// TwinCAT 3 PLC project TF3820StandalonePLC
// ProgramVersion: 3.1.4026.20
// libraries:
//   Tc2_Standard, * (Beckhoff Automation GmbH)
//   Tc2_System, * (Beckhoff Automation GmbH)
//   Tc3_MlServer, * (Beckhoff Automation GmbH)
// project tree:
//   DUTs/ E_TF3820StandaloneModelId.TcDUT, ST_FeedforwardInput.TcDUT, ST_FeedforwardOutput.TcDUT, ST_GruSequenceInput.TcDUT, ST_GruSequenceOutput.TcDUT, ST_HarmonicRegressionInput.TcDUT, ST_HarmonicRegressionOutput.TcDUT, ST_LstmSequenceInput.TcDUT, ST_LstmSequenceOutput.TcDUT, ST_PeriodicGruSequenceInput.TcDUT, ST_PeriodicGruSequenceOutput.TcDUT, ST_PeriodicLstmSequenceInput.TcDUT, ST_PeriodicLstmSequenceOutput.TcDUT, ST_PeriodicMlpInput.TcDUT, ST_PeriodicMlpOutput.TcDUT, ST_PeriodicMlpHarmonicInput.TcDUT, ST_PeriodicMlpHarmonicOutput.TcDUT, ST_PeriodicTemporalConvolutionInput.TcDUT, ST_PeriodicTemporalConvolutionOutput.TcDUT, ST_RcimTrack1Input.TcDUT, ST_RcimTrack1Output.TcDUT, ST_ResidualHarmonicGruSequenceDense240Input.TcDUT, ST_ResidualHarmonicGruSequenceDense240Output.TcDUT, ST_ResidualHarmonicGruSequenceDense360Input.TcDUT, ST_ResidualHarmonicGruSequenceDense360Output.TcDUT, ST_ResidualHarmonicGruSequenceSparseRcimInput.TcDUT, ST_ResidualHarmonicGruSequenceSparseRcimOutput.TcDUT, ST_ResidualHarmonicLstmSequenceDense240Input.TcDUT, ST_ResidualHarmonicLstmSequenceDense240Output.TcDUT, ST_ResidualHarmonicLstmSequenceDense360Input.TcDUT, ST_ResidualHarmonicLstmSequenceDense360Output.TcDUT, ST_ResidualHarmonicLstmSequenceSparseRcimInput.TcDUT, ST_ResidualHarmonicLstmSequenceSparseRcimOutput.TcDUT, ST_ResidualHarmonicMlpInput.TcDUT, ST_ResidualHarmonicMlpOutput.TcDUT, ST_TemporalConvolutionInput.TcDUT, ST_TemporalConvolutionOutput.TcDUT, ST_TreeInput.TcDUT, ST_TreeOutput.TcDUT, ST_Wave31SequentialResidualOffsetProbeInput.TcDUT, ST_Wave31SequentialResidualOffsetProbeOutput.TcDUT, ST_Wave32CleanSequentialResidualOffsetInput.TcDUT, ST_Wave32CleanSequentialResidualOffsetOutput.TcDUT, ST_Wave32HarmonicResidualOffsetInput.TcDUT, ST_Wave32HarmonicResidualOffsetOutput.TcDUT, ST_Wave33CurveAwarePointwiseControlInput.TcDUT, ST_Wave33CurveAwarePointwiseControlOutput.TcDUT, ST_Wave33FullCurveCompositeInput.TcDUT, ST_Wave33FullCurveCompositeOutput.TcDUT, ST_Wave33RawCenteredShapeCurveAwareInput.TcDUT, ST_Wave33RawCenteredShapeCurveAwareOutput.TcDUT, ST_Wave33RawOffsetCurveAwareInput.TcDUT, ST_Wave33RawOffsetCurveAwareOutput.TcDUT, ST_Wave41LogCoshRobustLossInput.TcDUT, ST_Wave41LogCoshRobustLossOutput.TcDUT, ST_Wave41MaeRobustLossInput.TcDUT, ST_Wave41MaeRobustLossOutput.TcDUT, ST_Wave41SmoothL1RobustLossInput.TcDUT, ST_Wave41SmoothL1RobustLossOutput.TcDUT, ST_Wave42GaussianNllInput.TcDUT, ST_Wave42GaussianNllOutput.TcDUT, ST_Wave42QuantileP10P50P90Input.TcDUT, ST_Wave42QuantileP10P50P90Output.TcDUT, ST_Wave43MixtureDensityK2Input.TcDUT, ST_Wave43MixtureDensityK2Output.TcDUT, ST_Wave43MixtureDensityK3Input.TcDUT, ST_Wave43MixtureDensityK3Output.TcDUT, ST_Wave44CausalTcnLatentOffsetResidualInput.TcDUT, ST_Wave44CausalTcnLatentOffsetResidualOutput.TcDUT, ST_Wave44GruLatentOffsetResidualInput.TcDUT, ST_Wave44GruLatentOffsetResidualOutput.TcDUT, ST_Wave51HarmonicPriorPointwiseControlInput.TcDUT, ST_Wave51HarmonicPriorPointwiseControlOutput.TcDUT, ST_Wave51HarmonicPriorSmoothL1StructuredInput.TcDUT, ST_Wave51HarmonicPriorSmoothL1StructuredOutput.TcDUT
//   / PlcTask_TF3820Standalone.TcTTO
//   POUs/ FB_FeedforwardTf3820Runner.TcPOU, FB_GruSequenceTf3820Runner.TcPOU, FB_HarmonicRegressionTf3820Runner.TcPOU, FB_LstmSequenceTf3820Runner.TcPOU, FB_PeriodicGruSequenceTf3820Runner.TcPOU, FB_PeriodicLstmSequenceTf3820Runner.TcPOU, FB_PeriodicMlpTf3820Runner.TcPOU, FB_PeriodicMlpHarmonicTf3820Runner.TcPOU, FB_PeriodicTemporalConvolutionTf3820Runner.TcPOU, FB_RcimTrack1Tf3820Runner.TcPOU, FB_ResidualHarmonicGruSequenceDense240Tf3820Runner.TcPOU, FB_ResidualHarmonicGruSequenceDense360Tf3820Runner.TcPOU, FB_ResidualHarmonicGruSequenceSparseRcimTf3820Runner.TcPOU, FB_ResidualHarmonicLstmSequenceDense240Tf3820Runner.TcPOU, FB_ResidualHarmonicLstmSequenceDense360Tf3820Runner.TcPOU, FB_ResidualHarmonicLstmSequenceSparseRcimTf3820Runner.TcPOU, FB_ResidualHarmonicMlpTf3820Runner.TcPOU, FB_TemporalConvolutionTf3820Runner.TcPOU, FB_TreeTf3820Runner.TcPOU, FB_Wave31SequentialResidualOffsetProbeTf3820Runner.TcPOU, FB_Wave32CleanSequentialResidualOffsetTf3820Runner.TcPOU, FB_Wave32HarmonicResidualOffsetTf3820Runner.TcPOU, FB_Wave33CurveAwarePointwiseControlTf3820Runner.TcPOU, FB_Wave33FullCurveCompositeTf3820Runner.TcPOU, FB_Wave33RawCenteredShapeCurveAwareTf3820Runner.TcPOU, FB_Wave33RawOffsetCurveAwareTf3820Runner.TcPOU, FB_Wave41LogCoshRobustLossTf3820Runner.TcPOU, FB_Wave41MaeRobustLossTf3820Runner.TcPOU, FB_Wave41SmoothL1RobustLossTf3820Runner.TcPOU, FB_Wave42GaussianNllTf3820Runner.TcPOU, FB_Wave42QuantileP10P50P90Tf3820Runner.TcPOU, FB_Wave43MixtureDensityK2Tf3820Runner.TcPOU, FB_Wave43MixtureDensityK3Tf3820Runner.TcPOU, FB_Wave44CausalTcnLatentOffsetResidualTf3820Runner.TcPOU, FB_Wave44GruLatentOffsetResidualTf3820Runner.TcPOU, FB_Wave51HarmonicPriorPointwiseControlTf3820Runner.TcPOU, FB_Wave51HarmonicPriorSmoothL1StructuredTf3820Runner.TcPOU, P_TF3820StandaloneModelTest.TcPOU
// real-time tasks:
//   TASK PlcTask_TF3820Standalone: cycle T#1ms, priority 10, ADS port 350

CONFIGURATION TF3820StandalonePLC
    RESOURCE PLC ON TwinCAT3
        TASK PlcTask_TF3820Standalone(INTERVAL := T#1ms, PRIORITY := 10);
        PROGRAM P_TF3820StandaloneModelTest WITH PlcTask_TF3820Standalone : P_TF3820StandaloneModelTest;
    END_RESOURCE
END_CONFIGURATION

// ---- DUTs/E_TF3820StandaloneModelId.TcDUT
{attribute 'qualified_only'}
{attribute 'strict'}
TYPE E_TF3820StandaloneModelId :
(
	Model_Feedforward := 0,
	Model_Gru_Sequence := 1,
	Model_Harmonic_Regression := 2,
	Model_Lstm_Sequence := 3,
	Model_Periodic_Gru_Sequence := 4,
	Model_Periodic_Lstm_Sequence := 5,
	Model_Periodic_Mlp := 6,
	Model_Periodic_Mlp_Harmonic := 7,
	Model_Periodic_Temporal_Convolution := 8,
	Model_Rcim_Track1 := 9,
	Model_Residual_Harmonic_Gru_Sequence_Dense240 := 10,
	Model_Residual_Harmonic_Gru_Sequence_Dense360 := 11,
	Model_Residual_Harmonic_Gru_Sequence_Sparse_Rcim := 12,
	Model_Residual_Harmonic_Lstm_Sequence_Dense240 := 13,
	Model_Residual_Harmonic_Lstm_Sequence_Dense360 := 14,
	Model_Residual_Harmonic_Lstm_Sequence_Sparse_Rcim := 15,
	Model_Residual_Harmonic_Mlp := 16,
	Model_Temporal_Convolution := 17,
	Model_Tree := 18,
	Model_Wave3_1_Sequential_Residual_Offset_Probe := 19,
	Model_Wave3_2_Clean_Sequential_Residual_Offset := 20,
	Model_Wave3_2_Harmonic_Residual_Offset := 21,
	Model_Wave3_3_Curve_Aware_Pointwise_Control := 22,
	Model_Wave3_3_Full_Curve_Composite := 23,
	Model_Wave3_3_Raw_Centered_Shape_Curve_Aware := 24,
	Model_Wave3_3_Raw_Offset_Curve_Aware := 25,
	Model_Wave4_1_Log_Cosh_Robust_Loss := 26,
	Model_Wave4_1_Mae_Robust_Loss := 27,
	Model_Wave4_1_Smooth_L1_Robust_Loss := 28,
	Model_Wave4_2_Gaussian_Nll := 29,
	Model_Wave4_2_Quantile_P10_P50_P90 := 30,
	Model_Wave4_3_Mixture_Density_K2 := 31,
	Model_Wave4_3_Mixture_Density_K3 := 32,
	Model_Wave4_4_Causal_Tcn_Latent_Offset_Residual := 33,
	Model_Wave4_4_Gru_Latent_Offset_Residual := 34,
	Model_Wave5_1_Harmonic_Prior_Pointwise_Control := 35,
	Model_Wave5_1_Harmonic_Prior_Smooth_L1_Structured := 36
);
END_TYPE

// ---- DUTs/ST_FeedforwardInput.TcDUT
TYPE ST_FeedforwardInput :
STRUCT

	{attribute 'hide'} _header_DO_NOT_CHANGE : ARRAY[0..63] OF SINT := [-1,-112,120,86,52,18,-1,-1,1,-1,0,0,-1,-1,-112,-112,61,-49,110,-13,101,63,-28,35,-75,-48,62,84,75,113,93,86,13,-100,61,-11,-76,-124,91,74,-32,110,127,-106,67,10,-85,-84,84,0,0,0,0,0,0,0,0,0,0,0,0,0,0,0];
	in_input_tensor : ARRAY[0..0,0..4] OF REAL;

END_STRUCT
END_TYPE

// ---- DUTs/ST_FeedforwardOutput.TcDUT
TYPE ST_FeedforwardOutput :
STRUCT

	{attribute 'hide'} _header_DO_NOT_CHANGE : ARRAY[0..63] OF SINT := [-1,-112,120,86,52,18,-1,-1,1,-1,0,0,-1,-1,-112,-112,-35,24,-50,75,-65,96,-121,123,127,87,61,127,-39,-108,16,-70,120,-89,-28,78,-43,26,-32,-7,81,19,29,-89,-55,3,43,2,68,0,0,0,0,0,0,0,0,0,0,0,0,0,0,0];
	out_prediction_tensor : ARRAY[0..0,0..0] OF REAL;

END_STRUCT
END_TYPE

// ---- DUTs/ST_GruSequenceInput.TcDUT
TYPE ST_GruSequenceInput :
STRUCT

	{attribute 'hide'} _header_DO_NOT_CHANGE : ARRAY[0..63] OF SINT := [-1,-112,120,86,52,18,-1,-1,1,-1,0,0,-1,-1,-112,-112,76,-37,-101,-100,-56,125,72,-20,-8,-106,39,-43,33,76,57,117,-100,-22,-66,-55,64,-24,-107,-56,26,-38,-68,-13,105,114,16,-98,-44,2,0,0,0,0,0,0,0,0,0,0,0,0,0,0];
	in_input_tensor : ARRAY[0..0,0..32,0..4] OF REAL;

END_STRUCT
END_TYPE

// ---- DUTs/ST_GruSequenceOutput.TcDUT
TYPE ST_GruSequenceOutput :
STRUCT

	{attribute 'hide'} _header_DO_NOT_CHANGE : ARRAY[0..63] OF SINT := [-1,-112,120,86,52,18,-1,-1,1,-1,0,0,-1,-1,-112,-112,-35,24,-50,75,-65,96,-121,123,127,87,61,127,-39,-108,16,-70,120,-89,-28,78,-43,26,-32,-7,81,19,29,-89,-55,3,43,2,68,0,0,0,0,0,0,0,0,0,0,0,0,0,0,0];
	out_prediction_tensor : ARRAY[0..0,0..0] OF REAL;

END_STRUCT
END_TYPE

// ---- DUTs/ST_HarmonicRegressionInput.TcDUT
TYPE ST_HarmonicRegressionInput :
STRUCT

	{attribute 'hide'} _header_DO_NOT_CHANGE : ARRAY[0..63] OF SINT := [-1,-112,120,86,52,18,-1,-1,1,-1,0,0,-1,-1,-112,-112,61,-49,110,-13,101,63,-28,35,-75,-48,62,84,75,113,93,86,13,-100,61,-11,-76,-124,91,74,-32,110,127,-106,67,10,-85,-84,84,0,0,0,0,0,0,0,0,0,0,0,0,0,0,0];
	in_input_tensor : ARRAY[0..0,0..4] OF REAL;

END_STRUCT
END_TYPE

// ---- DUTs/ST_HarmonicRegressionOutput.TcDUT
TYPE ST_HarmonicRegressionOutput :
STRUCT

	{attribute 'hide'} _header_DO_NOT_CHANGE : ARRAY[0..63] OF SINT := [-1,-112,120,86,52,18,-1,-1,1,-1,0,0,-1,-1,-112,-112,-35,24,-50,75,-65,96,-121,123,127,87,61,127,-39,-108,16,-70,120,-89,-28,78,-43,26,-32,-7,81,19,29,-89,-55,3,43,2,68,0,0,0,0,0,0,0,0,0,0,0,0,0,0,0];
	out_prediction_tensor : ARRAY[0..0,0..0] OF REAL;

END_STRUCT
END_TYPE

// ---- DUTs/ST_LstmSequenceInput.TcDUT
TYPE ST_LstmSequenceInput :
STRUCT

	{attribute 'hide'} _header_DO_NOT_CHANGE : ARRAY[0..63] OF SINT := [-1,-112,120,86,52,18,-1,-1,1,-1,0,0,-1,-1,-112,-112,76,-37,-101,-100,-56,125,72,-20,-8,-106,39,-43,33,76,57,117,-100,-22,-66,-55,64,-24,-107,-56,26,-38,-68,-13,105,114,16,-98,-44,2,0,0,0,0,0,0,0,0,0,0,0,0,0,0];
	in_input_tensor : ARRAY[0..0,0..32,0..4] OF REAL;

END_STRUCT
END_TYPE

// ---- DUTs/ST_LstmSequenceOutput.TcDUT
TYPE ST_LstmSequenceOutput :
STRUCT

	{attribute 'hide'} _header_DO_NOT_CHANGE : ARRAY[0..63] OF SINT := [-1,-112,120,86,52,18,-1,-1,1,-1,0,0,-1,-1,-112,-112,-35,24,-50,75,-65,96,-121,123,127,87,61,127,-39,-108,16,-70,120,-89,-28,78,-43,26,-32,-7,81,19,29,-89,-55,3,43,2,68,0,0,0,0,0,0,0,0,0,0,0,0,0,0,0];
	out_prediction_tensor : ARRAY[0..0,0..0] OF REAL;

END_STRUCT
END_TYPE

// ---- DUTs/ST_PeriodicGruSequenceInput.TcDUT
TYPE ST_PeriodicGruSequenceInput :
STRUCT

	{attribute 'hide'} _header_DO_NOT_CHANGE : ARRAY[0..63] OF SINT := [-1,-112,120,86,52,18,-1,-1,1,-1,0,0,-1,-1,-112,-112,76,-37,-101,-100,-56,125,72,-20,-8,-106,39,-43,33,76,57,117,-100,-22,-66,-55,64,-24,-107,-56,26,-38,-68,-13,105,114,16,-98,-44,2,0,0,0,0,0,0,0,0,0,0,0,0,0,0];
	in_input_tensor : ARRAY[0..0,0..32,0..4] OF REAL;

END_STRUCT
END_TYPE

// ---- DUTs/ST_PeriodicGruSequenceOutput.TcDUT
TYPE ST_PeriodicGruSequenceOutput :
STRUCT

	{attribute 'hide'} _header_DO_NOT_CHANGE : ARRAY[0..63] OF SINT := [-1,-112,120,86,52,18,-1,-1,1,-1,0,0,-1,-1,-112,-112,-35,24,-50,75,-65,96,-121,123,127,87,61,127,-39,-108,16,-70,120,-89,-28,78,-43,26,-32,-7,81,19,29,-89,-55,3,43,2,68,0,0,0,0,0,0,0,0,0,0,0,0,0,0,0];
	out_prediction_tensor : ARRAY[0..0,0..0] OF REAL;

END_STRUCT
END_TYPE

// ---- DUTs/ST_PeriodicLstmSequenceInput.TcDUT
TYPE ST_PeriodicLstmSequenceInput :
STRUCT

	{attribute 'hide'} _header_DO_NOT_CHANGE : ARRAY[0..63] OF SINT := [-1,-112,120,86,52,18,-1,-1,1,-1,0,0,-1,-1,-112,-112,76,-37,-101,-100,-56,125,72,-20,-8,-106,39,-43,33,76,57,117,-100,-22,-66,-55,64,-24,-107,-56,26,-38,-68,-13,105,114,16,-98,-44,2,0,0,0,0,0,0,0,0,0,0,0,0,0,0];
	in_input_tensor : ARRAY[0..0,0..32,0..4] OF REAL;

END_STRUCT
END_TYPE

// ---- DUTs/ST_PeriodicLstmSequenceOutput.TcDUT
TYPE ST_PeriodicLstmSequenceOutput :
STRUCT

	{attribute 'hide'} _header_DO_NOT_CHANGE : ARRAY[0..63] OF SINT := [-1,-112,120,86,52,18,-1,-1,1,-1,0,0,-1,-1,-112,-112,-35,24,-50,75,-65,96,-121,123,127,87,61,127,-39,-108,16,-70,120,-89,-28,78,-43,26,-32,-7,81,19,29,-89,-55,3,43,2,68,0,0,0,0,0,0,0,0,0,0,0,0,0,0,0];
	out_prediction_tensor : ARRAY[0..0,0..0] OF REAL;

END_STRUCT
END_TYPE

// ---- DUTs/ST_PeriodicMlpInput.TcDUT
TYPE ST_PeriodicMlpInput :
STRUCT

	{attribute 'hide'} _header_DO_NOT_CHANGE : ARRAY[0..63] OF SINT := [-1,-112,120,86,52,18,-1,-1,1,-1,0,0,-1,-1,-112,-112,61,-49,110,-13,101,63,-28,35,-75,-48,62,84,75,113,93,86,13,-100,61,-11,-76,-124,91,74,-32,110,127,-106,67,10,-85,-84,84,0,0,0,0,0,0,0,0,0,0,0,0,0,0,0];
	in_input_tensor : ARRAY[0..0,0..4] OF REAL;

END_STRUCT
END_TYPE

// ---- DUTs/ST_PeriodicMlpOutput.TcDUT
TYPE ST_PeriodicMlpOutput :
STRUCT

	{attribute 'hide'} _header_DO_NOT_CHANGE : ARRAY[0..63] OF SINT := [-1,-112,120,86,52,18,-1,-1,1,-1,0,0,-1,-1,-112,-112,-35,24,-50,75,-65,96,-121,123,127,87,61,127,-39,-108,16,-70,120,-89,-28,78,-43,26,-32,-7,81,19,29,-89,-55,3,43,2,68,0,0,0,0,0,0,0,0,0,0,0,0,0,0,0];
	out_prediction_tensor : ARRAY[0..0,0..0] OF REAL;

END_STRUCT
END_TYPE

// ---- DUTs/ST_PeriodicMlpHarmonicInput.TcDUT
TYPE ST_PeriodicMlpHarmonicInput :
STRUCT

	{attribute 'hide'} _header_DO_NOT_CHANGE : ARRAY[0..63] OF SINT := [-1,-112,120,86,52,18,-1,-1,1,-1,0,0,-1,-1,-112,-112,61,-49,110,-13,101,63,-28,35,-75,-48,62,84,75,113,93,86,13,-100,61,-11,-76,-124,91,74,-32,110,127,-106,67,10,-85,-84,84,0,0,0,0,0,0,0,0,0,0,0,0,0,0,0];
	in_input_tensor : ARRAY[0..0,0..4] OF REAL;

END_STRUCT
END_TYPE

// ---- DUTs/ST_PeriodicMlpHarmonicOutput.TcDUT
TYPE ST_PeriodicMlpHarmonicOutput :
STRUCT

	{attribute 'hide'} _header_DO_NOT_CHANGE : ARRAY[0..63] OF SINT := [-1,-112,120,86,52,18,-1,-1,1,-1,0,0,-1,-1,-112,-112,-35,24,-50,75,-65,96,-121,123,127,87,61,127,-39,-108,16,-70,120,-89,-28,78,-43,26,-32,-7,81,19,29,-89,-55,3,43,2,68,0,0,0,0,0,0,0,0,0,0,0,0,0,0,0];
	out_prediction_tensor : ARRAY[0..0,0..0] OF REAL;

END_STRUCT
END_TYPE

// ---- DUTs/ST_PeriodicTemporalConvolutionInput.TcDUT
TYPE ST_PeriodicTemporalConvolutionInput :
STRUCT

	{attribute 'hide'} _header_DO_NOT_CHANGE : ARRAY[0..63] OF SINT := [-1,-112,120,86,52,18,-1,-1,1,-1,0,0,-1,-1,-112,-112,76,-37,-101,-100,-56,125,72,-20,-8,-106,39,-43,33,76,57,117,-100,-22,-66,-55,64,-24,-107,-56,26,-38,-68,-13,105,114,16,-98,-44,2,0,0,0,0,0,0,0,0,0,0,0,0,0,0];
	in_input_tensor : ARRAY[0..0,0..32,0..4] OF REAL;

END_STRUCT
END_TYPE

// ---- DUTs/ST_PeriodicTemporalConvolutionOutput.TcDUT
TYPE ST_PeriodicTemporalConvolutionOutput :
STRUCT

	{attribute 'hide'} _header_DO_NOT_CHANGE : ARRAY[0..63] OF SINT := [-1,-112,120,86,52,18,-1,-1,1,-1,0,0,-1,-1,-112,-112,-35,24,-50,75,-65,96,-121,123,127,87,61,127,-39,-108,16,-70,120,-89,-28,78,-43,26,-32,-7,81,19,29,-89,-55,3,43,2,68,0,0,0,0,0,0,0,0,0,0,0,0,0,0,0];
	out_prediction_tensor : ARRAY[0..0,0..0] OF REAL;

END_STRUCT
END_TYPE

// ---- DUTs/ST_RcimTrack1Input.TcDUT
TYPE ST_RcimTrack1Input :
STRUCT

	{attribute 'hide'} _header_DO_NOT_CHANGE : ARRAY[0..63] OF SINT := [-1,-112,120,86,52,18,-1,-1,1,-1,0,0,-1,-1,-112,-112,65,64,108,85,118,21,-37,1,110,122,-102,19,93,-117,-35,-43,3,-45,33,-52,25,-24,90,7,83,36,22,5,-43,-65,-103,-61,76,0,0,0,0,0,0,0,0,0,0,0,0,0,0,0];
	in_float_input : ARRAY[0..0,0..2] OF REAL;

END_STRUCT
END_TYPE

// ---- DUTs/ST_RcimTrack1Output.TcDUT
TYPE ST_RcimTrack1Output :
STRUCT

	{attribute 'hide'} _header_DO_NOT_CHANGE : ARRAY[0..63] OF SINT := [-1,-112,120,86,52,18,-1,-1,1,-1,0,0,-1,-1,-112,-112,-35,24,-50,75,-65,96,-121,123,127,87,61,127,-39,-108,16,-70,120,-89,-28,78,-43,26,-32,-7,81,19,29,-89,-55,3,43,2,68,0,0,0,0,0,0,0,0,0,0,0,0,0,0,0];
	out_variable : ARRAY[0..0,0..0] OF REAL;

END_STRUCT
END_TYPE

// ---- DUTs/ST_ResidualHarmonicGruSequenceDense240Input.TcDUT
TYPE ST_ResidualHarmonicGruSequenceDense240Input :
STRUCT

	{attribute 'hide'} _header_DO_NOT_CHANGE : ARRAY[0..63] OF SINT := [-1,-112,120,86,52,18,-1,-1,1,-1,0,0,-1,-1,-112,-112,76,-37,-101,-100,-56,125,72,-20,-8,-106,39,-43,33,76,57,117,-100,-22,-66,-55,64,-24,-107,-56,26,-38,-68,-13,105,114,16,-98,-44,2,0,0,0,0,0,0,0,0,0,0,0,0,0,0];
	in_input_tensor : ARRAY[0..0,0..32,0..4] OF REAL;

END_STRUCT
END_TYPE

// ---- DUTs/ST_ResidualHarmonicGruSequenceDense240Output.TcDUT
TYPE ST_ResidualHarmonicGruSequenceDense240Output :
STRUCT

	{attribute 'hide'} _header_DO_NOT_CHANGE : ARRAY[0..63] OF SINT := [-1,-112,120,86,52,18,-1,-1,1,-1,0,0,-1,-1,-112,-112,-35,24,-50,75,-65,96,-121,123,127,87,61,127,-39,-108,16,-70,120,-89,-28,78,-43,26,-32,-7,81,19,29,-89,-55,3,43,2,68,0,0,0,0,0,0,0,0,0,0,0,0,0,0,0];
	out_prediction_tensor : ARRAY[0..0,0..0] OF REAL;

END_STRUCT
END_TYPE

// ---- DUTs/ST_ResidualHarmonicGruSequenceDense360Input.TcDUT
TYPE ST_ResidualHarmonicGruSequenceDense360Input :
STRUCT

	{attribute 'hide'} _header_DO_NOT_CHANGE : ARRAY[0..63] OF SINT := [-1,-112,120,86,52,18,-1,-1,1,-1,0,0,-1,-1,-112,-112,76,-37,-101,-100,-56,125,72,-20,-8,-106,39,-43,33,76,57,117,-100,-22,-66,-55,64,-24,-107,-56,26,-38,-68,-13,105,114,16,-98,-44,2,0,0,0,0,0,0,0,0,0,0,0,0,0,0];
	in_input_tensor : ARRAY[0..0,0..32,0..4] OF REAL;

END_STRUCT
END_TYPE

// ---- DUTs/ST_ResidualHarmonicGruSequenceDense360Output.TcDUT
TYPE ST_ResidualHarmonicGruSequenceDense360Output :
STRUCT

	{attribute 'hide'} _header_DO_NOT_CHANGE : ARRAY[0..63] OF SINT := [-1,-112,120,86,52,18,-1,-1,1,-1,0,0,-1,-1,-112,-112,-35,24,-50,75,-65,96,-121,123,127,87,61,127,-39,-108,16,-70,120,-89,-28,78,-43,26,-32,-7,81,19,29,-89,-55,3,43,2,68,0,0,0,0,0,0,0,0,0,0,0,0,0,0,0];
	out_prediction_tensor : ARRAY[0..0,0..0] OF REAL;

END_STRUCT
END_TYPE

// ---- DUTs/ST_ResidualHarmonicGruSequenceSparseRcimInput.TcDUT
TYPE ST_ResidualHarmonicGruSequenceSparseRcimInput :
STRUCT

	{attribute 'hide'} _header_DO_NOT_CHANGE : ARRAY[0..63] OF SINT := [-1,-112,120,86,52,18,-1,-1,1,-1,0,0,-1,-1,-112,-112,76,-37,-101,-100,-56,125,72,-20,-8,-106,39,-43,33,76,57,117,-100,-22,-66,-55,64,-24,-107,-56,26,-38,-68,-13,105,114,16,-98,-44,2,0,0,0,0,0,0,0,0,0,0,0,0,0,0];
	in_input_tensor : ARRAY[0..0,0..32,0..4] OF REAL;

END_STRUCT
END_TYPE

// ---- DUTs/ST_ResidualHarmonicGruSequenceSparseRcimOutput.TcDUT
TYPE ST_ResidualHarmonicGruSequenceSparseRcimOutput :
STRUCT

	{attribute 'hide'} _header_DO_NOT_CHANGE : ARRAY[0..63] OF SINT := [-1,-112,120,86,52,18,-1,-1,1,-1,0,0,-1,-1,-112,-112,-35,24,-50,75,-65,96,-121,123,127,87,61,127,-39,-108,16,-70,120,-89,-28,78,-43,26,-32,-7,81,19,29,-89,-55,3,43,2,68,0,0,0,0,0,0,0,0,0,0,0,0,0,0,0];
	out_prediction_tensor : ARRAY[0..0,0..0] OF REAL;

END_STRUCT
END_TYPE

// ---- DUTs/ST_ResidualHarmonicLstmSequenceDense240Input.TcDUT
TYPE ST_ResidualHarmonicLstmSequenceDense240Input :
STRUCT

	{attribute 'hide'} _header_DO_NOT_CHANGE : ARRAY[0..63] OF SINT := [-1,-112,120,86,52,18,-1,-1,1,-1,0,0,-1,-1,-112,-112,76,-37,-101,-100,-56,125,72,-20,-8,-106,39,-43,33,76,57,117,-100,-22,-66,-55,64,-24,-107,-56,26,-38,-68,-13,105,114,16,-98,-44,2,0,0,0,0,0,0,0,0,0,0,0,0,0,0];
	in_input_tensor : ARRAY[0..0,0..32,0..4] OF REAL;

END_STRUCT
END_TYPE

// ---- DUTs/ST_ResidualHarmonicLstmSequenceDense240Output.TcDUT
TYPE ST_ResidualHarmonicLstmSequenceDense240Output :
STRUCT

	{attribute 'hide'} _header_DO_NOT_CHANGE : ARRAY[0..63] OF SINT := [-1,-112,120,86,52,18,-1,-1,1,-1,0,0,-1,-1,-112,-112,-35,24,-50,75,-65,96,-121,123,127,87,61,127,-39,-108,16,-70,120,-89,-28,78,-43,26,-32,-7,81,19,29,-89,-55,3,43,2,68,0,0,0,0,0,0,0,0,0,0,0,0,0,0,0];
	out_prediction_tensor : ARRAY[0..0,0..0] OF REAL;

END_STRUCT
END_TYPE

// ---- DUTs/ST_ResidualHarmonicLstmSequenceDense360Input.TcDUT
TYPE ST_ResidualHarmonicLstmSequenceDense360Input :
STRUCT

	{attribute 'hide'} _header_DO_NOT_CHANGE : ARRAY[0..63] OF SINT := [-1,-112,120,86,52,18,-1,-1,1,-1,0,0,-1,-1,-112,-112,76,-37,-101,-100,-56,125,72,-20,-8,-106,39,-43,33,76,57,117,-100,-22,-66,-55,64,-24,-107,-56,26,-38,-68,-13,105,114,16,-98,-44,2,0,0,0,0,0,0,0,0,0,0,0,0,0,0];
	in_input_tensor : ARRAY[0..0,0..32,0..4] OF REAL;

END_STRUCT
END_TYPE

// ---- DUTs/ST_ResidualHarmonicLstmSequenceDense360Output.TcDUT
TYPE ST_ResidualHarmonicLstmSequenceDense360Output :
STRUCT

	{attribute 'hide'} _header_DO_NOT_CHANGE : ARRAY[0..63] OF SINT := [-1,-112,120,86,52,18,-1,-1,1,-1,0,0,-1,-1,-112,-112,-35,24,-50,75,-65,96,-121,123,127,87,61,127,-39,-108,16,-70,120,-89,-28,78,-43,26,-32,-7,81,19,29,-89,-55,3,43,2,68,0,0,0,0,0,0,0,0,0,0,0,0,0,0,0];
	out_prediction_tensor : ARRAY[0..0,0..0] OF REAL;

END_STRUCT
END_TYPE

// ---- DUTs/ST_ResidualHarmonicLstmSequenceSparseRcimInput.TcDUT
TYPE ST_ResidualHarmonicLstmSequenceSparseRcimInput :
STRUCT

	{attribute 'hide'} _header_DO_NOT_CHANGE : ARRAY[0..63] OF SINT := [-1,-112,120,86,52,18,-1,-1,1,-1,0,0,-1,-1,-112,-112,76,-37,-101,-100,-56,125,72,-20,-8,-106,39,-43,33,76,57,117,-100,-22,-66,-55,64,-24,-107,-56,26,-38,-68,-13,105,114,16,-98,-44,2,0,0,0,0,0,0,0,0,0,0,0,0,0,0];
	in_input_tensor : ARRAY[0..0,0..32,0..4] OF REAL;

END_STRUCT
END_TYPE

// ---- DUTs/ST_ResidualHarmonicLstmSequenceSparseRcimOutput.TcDUT
TYPE ST_ResidualHarmonicLstmSequenceSparseRcimOutput :
STRUCT

	{attribute 'hide'} _header_DO_NOT_CHANGE : ARRAY[0..63] OF SINT := [-1,-112,120,86,52,18,-1,-1,1,-1,0,0,-1,-1,-112,-112,-35,24,-50,75,-65,96,-121,123,127,87,61,127,-39,-108,16,-70,120,-89,-28,78,-43,26,-32,-7,81,19,29,-89,-55,3,43,2,68,0,0,0,0,0,0,0,0,0,0,0,0,0,0,0];
	out_prediction_tensor : ARRAY[0..0,0..0] OF REAL;

END_STRUCT
END_TYPE

// ---- DUTs/ST_ResidualHarmonicMlpInput.TcDUT
TYPE ST_ResidualHarmonicMlpInput :
STRUCT

	{attribute 'hide'} _header_DO_NOT_CHANGE : ARRAY[0..63] OF SINT := [-1,-112,120,86,52,18,-1,-1,1,-1,0,0,-1,-1,-112,-112,61,-49,110,-13,101,63,-28,35,-75,-48,62,84,75,113,93,86,13,-100,61,-11,-76,-124,91,74,-32,110,127,-106,67,10,-85,-84,84,0,0,0,0,0,0,0,0,0,0,0,0,0,0,0];
	in_input_tensor : ARRAY[0..0,0..4] OF REAL;

END_STRUCT
END_TYPE

// ---- DUTs/ST_ResidualHarmonicMlpOutput.TcDUT
TYPE ST_ResidualHarmonicMlpOutput :
STRUCT

	{attribute 'hide'} _header_DO_NOT_CHANGE : ARRAY[0..63] OF SINT := [-1,-112,120,86,52,18,-1,-1,1,-1,0,0,-1,-1,-112,-112,-35,24,-50,75,-65,96,-121,123,127,87,61,127,-39,-108,16,-70,120,-89,-28,78,-43,26,-32,-7,81,19,29,-89,-55,3,43,2,68,0,0,0,0,0,0,0,0,0,0,0,0,0,0,0];
	out_prediction_tensor : ARRAY[0..0,0..0] OF REAL;

END_STRUCT
END_TYPE

// ---- DUTs/ST_TemporalConvolutionInput.TcDUT
TYPE ST_TemporalConvolutionInput :
STRUCT

	{attribute 'hide'} _header_DO_NOT_CHANGE : ARRAY[0..63] OF SINT := [-1,-112,120,86,52,18,-1,-1,1,-1,0,0,-1,-1,-112,-112,76,-37,-101,-100,-56,125,72,-20,-8,-106,39,-43,33,76,57,117,-100,-22,-66,-55,64,-24,-107,-56,26,-38,-68,-13,105,114,16,-98,-44,2,0,0,0,0,0,0,0,0,0,0,0,0,0,0];
	in_input_tensor : ARRAY[0..0,0..32,0..4] OF REAL;

END_STRUCT
END_TYPE

// ---- DUTs/ST_TemporalConvolutionOutput.TcDUT
TYPE ST_TemporalConvolutionOutput :
STRUCT

	{attribute 'hide'} _header_DO_NOT_CHANGE : ARRAY[0..63] OF SINT := [-1,-112,120,86,52,18,-1,-1,1,-1,0,0,-1,-1,-112,-112,-35,24,-50,75,-65,96,-121,123,127,87,61,127,-39,-108,16,-70,120,-89,-28,78,-43,26,-32,-7,81,19,29,-89,-55,3,43,2,68,0,0,0,0,0,0,0,0,0,0,0,0,0,0,0];
	out_prediction_tensor : ARRAY[0..0,0..0] OF REAL;

END_STRUCT
END_TYPE

// ---- DUTs/ST_TreeInput.TcDUT
TYPE ST_TreeInput :
STRUCT

	{attribute 'hide'} _header_DO_NOT_CHANGE : ARRAY[0..63] OF SINT := [-1,-112,120,86,52,18,-1,-1,1,-1,0,0,-1,-1,-112,-112,61,-49,110,-13,101,63,-28,35,-75,-48,62,84,75,113,93,86,13,-100,61,-11,-76,-124,91,74,-32,110,127,-106,67,10,-85,-84,84,0,0,0,0,0,0,0,0,0,0,0,0,0,0,0];
	in_float_input : ARRAY[0..0,0..4] OF REAL;

END_STRUCT
END_TYPE

// ---- DUTs/ST_TreeOutput.TcDUT
TYPE ST_TreeOutput :
STRUCT

	{attribute 'hide'} _header_DO_NOT_CHANGE : ARRAY[0..63] OF SINT := [-1,-112,120,86,52,18,-1,-1,1,-1,0,0,-1,-1,-112,-112,-35,24,-50,75,-65,96,-121,123,127,87,61,127,-39,-108,16,-70,120,-89,-28,78,-43,26,-32,-7,81,19,29,-89,-55,3,43,2,68,0,0,0,0,0,0,0,0,0,0,0,0,0,0,0];
	out_variable : ARRAY[0..0,0..0] OF REAL;

END_STRUCT
END_TYPE

// ---- DUTs/ST_Wave31SequentialResidualOffsetProbeInput.TcDUT
TYPE ST_Wave31SequentialResidualOffsetProbeInput :
STRUCT

	{attribute 'hide'} _header_DO_NOT_CHANGE : ARRAY[0..63] OF SINT := [-1,-112,120,86,52,18,-1,-1,1,-1,0,0,-1,-1,-112,-112,76,-37,-101,-100,-56,125,72,-20,-8,-106,39,-43,33,76,57,117,-100,-22,-66,-55,64,-24,-107,-56,26,-38,-68,-13,105,114,16,-98,-44,2,0,0,0,0,0,0,0,0,0,0,0,0,0,0];
	in_input_tensor : ARRAY[0..0,0..32,0..4] OF REAL;

END_STRUCT
END_TYPE

// ---- DUTs/ST_Wave31SequentialResidualOffsetProbeOutput.TcDUT
TYPE ST_Wave31SequentialResidualOffsetProbeOutput :
STRUCT

	{attribute 'hide'} _header_DO_NOT_CHANGE : ARRAY[0..63] OF SINT := [-1,-112,120,86,52,18,-1,-1,1,-1,0,0,-1,-1,-112,-112,-35,24,-50,75,-65,96,-121,123,127,87,61,127,-39,-108,16,-70,120,-89,-28,78,-43,26,-32,-7,81,19,29,-89,-55,3,43,2,68,0,0,0,0,0,0,0,0,0,0,0,0,0,0,0];
	out_prediction_tensor : ARRAY[0..0,0..0] OF REAL;

END_STRUCT
END_TYPE

// ---- DUTs/ST_Wave32CleanSequentialResidualOffsetInput.TcDUT
TYPE ST_Wave32CleanSequentialResidualOffsetInput :
STRUCT

	{attribute 'hide'} _header_DO_NOT_CHANGE : ARRAY[0..63] OF SINT := [-1,-112,120,86,52,18,-1,-1,1,-1,0,0,-1,-1,-112,-112,55,-22,8,-62,15,-11,-53,-120,-65,-26,40,-59,-103,80,20,5,37,-41,0,-16,-125,-33,-67,117,-59,70,-31,-53,-46,-33,-68,-19,80,2,0,0,0,0,0,0,0,0,0,0,0,0,0,0];
	in_input_tensor : ARRAY[0..0,0..32,0..3] OF REAL;

END_STRUCT
END_TYPE

// ---- DUTs/ST_Wave32CleanSequentialResidualOffsetOutput.TcDUT
TYPE ST_Wave32CleanSequentialResidualOffsetOutput :
STRUCT

	{attribute 'hide'} _header_DO_NOT_CHANGE : ARRAY[0..63] OF SINT := [-1,-112,120,86,52,18,-1,-1,1,-1,0,0,-1,-1,-112,-112,-35,24,-50,75,-65,96,-121,123,127,87,61,127,-39,-108,16,-70,120,-89,-28,78,-43,26,-32,-7,81,19,29,-89,-55,3,43,2,68,0,0,0,0,0,0,0,0,0,0,0,0,0,0,0];
	out_prediction_tensor : ARRAY[0..0,0..0] OF REAL;

END_STRUCT
END_TYPE

// ---- DUTs/ST_Wave32HarmonicResidualOffsetInput.TcDUT
TYPE ST_Wave32HarmonicResidualOffsetInput :
STRUCT

	{attribute 'hide'} _header_DO_NOT_CHANGE : ARRAY[0..63] OF SINT := [-1,-112,120,86,52,18,-1,-1,1,-1,0,0,-1,-1,-112,-112,55,-22,8,-62,15,-11,-53,-120,-65,-26,40,-59,-103,80,20,5,37,-41,0,-16,-125,-33,-67,117,-59,70,-31,-53,-46,-33,-68,-19,80,2,0,0,0,0,0,0,0,0,0,0,0,0,0,0];
	in_input_tensor : ARRAY[0..0,0..32,0..3] OF REAL;

END_STRUCT
END_TYPE

// ---- DUTs/ST_Wave32HarmonicResidualOffsetOutput.TcDUT
TYPE ST_Wave32HarmonicResidualOffsetOutput :
STRUCT

	{attribute 'hide'} _header_DO_NOT_CHANGE : ARRAY[0..63] OF SINT := [-1,-112,120,86,52,18,-1,-1,1,-1,0,0,-1,-1,-112,-112,-35,24,-50,75,-65,96,-121,123,127,87,61,127,-39,-108,16,-70,120,-89,-28,78,-43,26,-32,-7,81,19,29,-89,-55,3,43,2,68,0,0,0,0,0,0,0,0,0,0,0,0,0,0,0];
	out_prediction_tensor : ARRAY[0..0,0..0] OF REAL;

END_STRUCT
END_TYPE

// ---- DUTs/ST_Wave33CurveAwarePointwiseControlInput.TcDUT
TYPE ST_Wave33CurveAwarePointwiseControlInput :
STRUCT

	{attribute 'hide'} _header_DO_NOT_CHANGE : ARRAY[0..63] OF SINT := [-1,-112,120,86,52,18,-1,-1,1,-1,0,0,-1,-1,-112,-112,55,-22,8,-62,15,-11,-53,-120,-65,-26,40,-59,-103,80,20,5,37,-41,0,-16,-125,-33,-67,117,-59,70,-31,-53,-46,-33,-68,-19,80,2,0,0,0,0,0,0,0,0,0,0,0,0,0,0];
	in_input_tensor : ARRAY[0..0,0..32,0..3] OF REAL;

END_STRUCT
END_TYPE

// ---- DUTs/ST_Wave33CurveAwarePointwiseControlOutput.TcDUT
TYPE ST_Wave33CurveAwarePointwiseControlOutput :
STRUCT

	{attribute 'hide'} _header_DO_NOT_CHANGE : ARRAY[0..63] OF SINT := [-1,-112,120,86,52,18,-1,-1,1,-1,0,0,-1,-1,-112,-112,-35,24,-50,75,-65,96,-121,123,127,87,61,127,-39,-108,16,-70,120,-89,-28,78,-43,26,-32,-7,81,19,29,-89,-55,3,43,2,68,0,0,0,0,0,0,0,0,0,0,0,0,0,0,0];
	out_prediction_tensor : ARRAY[0..0,0..0] OF REAL;

END_STRUCT
END_TYPE

// ---- DUTs/ST_Wave33FullCurveCompositeInput.TcDUT
TYPE ST_Wave33FullCurveCompositeInput :
STRUCT

	{attribute 'hide'} _header_DO_NOT_CHANGE : ARRAY[0..63] OF SINT := [-1,-112,120,86,52,18,-1,-1,1,-1,0,0,-1,-1,-112,-112,55,-22,8,-62,15,-11,-53,-120,-65,-26,40,-59,-103,80,20,5,37,-41,0,-16,-125,-33,-67,117,-59,70,-31,-53,-46,-33,-68,-19,80,2,0,0,0,0,0,0,0,0,0,0,0,0,0,0];
	in_input_tensor : ARRAY[0..0,0..32,0..3] OF REAL;

END_STRUCT
END_TYPE

// ---- DUTs/ST_Wave33FullCurveCompositeOutput.TcDUT
TYPE ST_Wave33FullCurveCompositeOutput :
STRUCT

	{attribute 'hide'} _header_DO_NOT_CHANGE : ARRAY[0..63] OF SINT := [-1,-112,120,86,52,18,-1,-1,1,-1,0,0,-1,-1,-112,-112,-35,24,-50,75,-65,96,-121,123,127,87,61,127,-39,-108,16,-70,120,-89,-28,78,-43,26,-32,-7,81,19,29,-89,-55,3,43,2,68,0,0,0,0,0,0,0,0,0,0,0,0,0,0,0];
	out_prediction_tensor : ARRAY[0..0,0..0] OF REAL;

END_STRUCT
END_TYPE

// ---- DUTs/ST_Wave33RawCenteredShapeCurveAwareInput.TcDUT
TYPE ST_Wave33RawCenteredShapeCurveAwareInput :
STRUCT

	{attribute 'hide'} _header_DO_NOT_CHANGE : ARRAY[0..63] OF SINT := [-1,-112,120,86,52,18,-1,-1,1,-1,0,0,-1,-1,-112,-112,55,-22,8,-62,15,-11,-53,-120,-65,-26,40,-59,-103,80,20,5,37,-41,0,-16,-125,-33,-67,117,-59,70,-31,-53,-46,-33,-68,-19,80,2,0,0,0,0,0,0,0,0,0,0,0,0,0,0];
	in_input_tensor : ARRAY[0..0,0..32,0..3] OF REAL;

END_STRUCT
END_TYPE

// ---- DUTs/ST_Wave33RawCenteredShapeCurveAwareOutput.TcDUT
TYPE ST_Wave33RawCenteredShapeCurveAwareOutput :
STRUCT

	{attribute 'hide'} _header_DO_NOT_CHANGE : ARRAY[0..63] OF SINT := [-1,-112,120,86,52,18,-1,-1,1,-1,0,0,-1,-1,-112,-112,-35,24,-50,75,-65,96,-121,123,127,87,61,127,-39,-108,16,-70,120,-89,-28,78,-43,26,-32,-7,81,19,29,-89,-55,3,43,2,68,0,0,0,0,0,0,0,0,0,0,0,0,0,0,0];
	out_prediction_tensor : ARRAY[0..0,0..0] OF REAL;

END_STRUCT
END_TYPE

// ---- DUTs/ST_Wave33RawOffsetCurveAwareInput.TcDUT
TYPE ST_Wave33RawOffsetCurveAwareInput :
STRUCT

	{attribute 'hide'} _header_DO_NOT_CHANGE : ARRAY[0..63] OF SINT := [-1,-112,120,86,52,18,-1,-1,1,-1,0,0,-1,-1,-112,-112,55,-22,8,-62,15,-11,-53,-120,-65,-26,40,-59,-103,80,20,5,37,-41,0,-16,-125,-33,-67,117,-59,70,-31,-53,-46,-33,-68,-19,80,2,0,0,0,0,0,0,0,0,0,0,0,0,0,0];
	in_input_tensor : ARRAY[0..0,0..32,0..3] OF REAL;

END_STRUCT
END_TYPE

// ---- DUTs/ST_Wave33RawOffsetCurveAwareOutput.TcDUT
TYPE ST_Wave33RawOffsetCurveAwareOutput :
STRUCT

	{attribute 'hide'} _header_DO_NOT_CHANGE : ARRAY[0..63] OF SINT := [-1,-112,120,86,52,18,-1,-1,1,-1,0,0,-1,-1,-112,-112,-35,24,-50,75,-65,96,-121,123,127,87,61,127,-39,-108,16,-70,120,-89,-28,78,-43,26,-32,-7,81,19,29,-89,-55,3,43,2,68,0,0,0,0,0,0,0,0,0,0,0,0,0,0,0];
	out_prediction_tensor : ARRAY[0..0,0..0] OF REAL;

END_STRUCT
END_TYPE

// ---- DUTs/ST_Wave41LogCoshRobustLossInput.TcDUT
TYPE ST_Wave41LogCoshRobustLossInput :
STRUCT

	{attribute 'hide'} _header_DO_NOT_CHANGE : ARRAY[0..63] OF SINT := [-1,-112,120,86,52,18,-1,-1,1,-1,0,0,-1,-1,-112,-112,55,-22,8,-62,15,-11,-53,-120,-65,-26,40,-59,-103,80,20,5,37,-41,0,-16,-125,-33,-67,117,-59,70,-31,-53,-46,-33,-68,-19,80,2,0,0,0,0,0,0,0,0,0,0,0,0,0,0];
	in_input_tensor : ARRAY[0..0,0..32,0..3] OF REAL;

END_STRUCT
END_TYPE

// ---- DUTs/ST_Wave41LogCoshRobustLossOutput.TcDUT
TYPE ST_Wave41LogCoshRobustLossOutput :
STRUCT

	{attribute 'hide'} _header_DO_NOT_CHANGE : ARRAY[0..63] OF SINT := [-1,-112,120,86,52,18,-1,-1,1,-1,0,0,-1,-1,-112,-112,-35,24,-50,75,-65,96,-121,123,127,87,61,127,-39,-108,16,-70,120,-89,-28,78,-43,26,-32,-7,81,19,29,-89,-55,3,43,2,68,0,0,0,0,0,0,0,0,0,0,0,0,0,0,0];
	out_prediction_tensor : ARRAY[0..0,0..0] OF REAL;

END_STRUCT
END_TYPE

// ---- DUTs/ST_Wave41MaeRobustLossInput.TcDUT
TYPE ST_Wave41MaeRobustLossInput :
STRUCT

	{attribute 'hide'} _header_DO_NOT_CHANGE : ARRAY[0..63] OF SINT := [-1,-112,120,86,52,18,-1,-1,1,-1,0,0,-1,-1,-112,-112,55,-22,8,-62,15,-11,-53,-120,-65,-26,40,-59,-103,80,20,5,37,-41,0,-16,-125,-33,-67,117,-59,70,-31,-53,-46,-33,-68,-19,80,2,0,0,0,0,0,0,0,0,0,0,0,0,0,0];
	in_input_tensor : ARRAY[0..0,0..32,0..3] OF REAL;

END_STRUCT
END_TYPE

// ---- DUTs/ST_Wave41MaeRobustLossOutput.TcDUT
TYPE ST_Wave41MaeRobustLossOutput :
STRUCT

	{attribute 'hide'} _header_DO_NOT_CHANGE : ARRAY[0..63] OF SINT := [-1,-112,120,86,52,18,-1,-1,1,-1,0,0,-1,-1,-112,-112,-35,24,-50,75,-65,96,-121,123,127,87,61,127,-39,-108,16,-70,120,-89,-28,78,-43,26,-32,-7,81,19,29,-89,-55,3,43,2,68,0,0,0,0,0,0,0,0,0,0,0,0,0,0,0];
	out_prediction_tensor : ARRAY[0..0,0..0] OF REAL;

END_STRUCT
END_TYPE

// ---- DUTs/ST_Wave41SmoothL1RobustLossInput.TcDUT
TYPE ST_Wave41SmoothL1RobustLossInput :
STRUCT

	{attribute 'hide'} _header_DO_NOT_CHANGE : ARRAY[0..63] OF SINT := [-1,-112,120,86,52,18,-1,-1,1,-1,0,0,-1,-1,-112,-112,55,-22,8,-62,15,-11,-53,-120,-65,-26,40,-59,-103,80,20,5,37,-41,0,-16,-125,-33,-67,117,-59,70,-31,-53,-46,-33,-68,-19,80,2,0,0,0,0,0,0,0,0,0,0,0,0,0,0];
	in_input_tensor : ARRAY[0..0,0..32,0..3] OF REAL;

END_STRUCT
END_TYPE

// ---- DUTs/ST_Wave41SmoothL1RobustLossOutput.TcDUT
TYPE ST_Wave41SmoothL1RobustLossOutput :
STRUCT

	{attribute 'hide'} _header_DO_NOT_CHANGE : ARRAY[0..63] OF SINT := [-1,-112,120,86,52,18,-1,-1,1,-1,0,0,-1,-1,-112,-112,-35,24,-50,75,-65,96,-121,123,127,87,61,127,-39,-108,16,-70,120,-89,-28,78,-43,26,-32,-7,81,19,29,-89,-55,3,43,2,68,0,0,0,0,0,0,0,0,0,0,0,0,0,0,0];
	out_prediction_tensor : ARRAY[0..0,0..0] OF REAL;

END_STRUCT
END_TYPE

// ---- DUTs/ST_Wave42GaussianNllInput.TcDUT
TYPE ST_Wave42GaussianNllInput :
STRUCT

	{attribute 'hide'} _header_DO_NOT_CHANGE : ARRAY[0..63] OF SINT := [-1,-112,120,86,52,18,-1,-1,1,-1,0,0,-1,-1,-112,-112,55,-22,8,-62,15,-11,-53,-120,-65,-26,40,-59,-103,80,20,5,37,-41,0,-16,-125,-33,-67,117,-59,70,-31,-53,-46,-33,-68,-19,80,2,0,0,0,0,0,0,0,0,0,0,0,0,0,0];
	in_input_tensor : ARRAY[0..0,0..32,0..3] OF REAL;

END_STRUCT
END_TYPE

// ---- DUTs/ST_Wave42GaussianNllOutput.TcDUT
TYPE ST_Wave42GaussianNllOutput :
STRUCT

	{attribute 'hide'} _header_DO_NOT_CHANGE : ARRAY[0..63] OF SINT := [-1,-112,120,86,52,18,-1,-1,1,-1,0,0,-1,-1,-112,-112,-76,58,-78,-85,-19,63,-109,100,101,125,-3,4,95,-56,77,-55,-69,-73,-40,-53,-105,-37,77,13,46,113,-54,-50,18,2,-83,14,72,0,0,0,0,0,0,0,0,0,0,0,0,0,0,0];
	out_prediction_tensor : ARRAY[0..0,0..1] OF REAL;

END_STRUCT
END_TYPE

// ---- DUTs/ST_Wave42QuantileP10P50P90Input.TcDUT
TYPE ST_Wave42QuantileP10P50P90Input :
STRUCT

	{attribute 'hide'} _header_DO_NOT_CHANGE : ARRAY[0..63] OF SINT := [-1,-112,120,86,52,18,-1,-1,1,-1,0,0,-1,-1,-112,-112,55,-22,8,-62,15,-11,-53,-120,-65,-26,40,-59,-103,80,20,5,37,-41,0,-16,-125,-33,-67,117,-59,70,-31,-53,-46,-33,-68,-19,80,2,0,0,0,0,0,0,0,0,0,0,0,0,0,0];
	in_input_tensor : ARRAY[0..0,0..32,0..3] OF REAL;

END_STRUCT
END_TYPE

// ---- DUTs/ST_Wave42QuantileP10P50P90Output.TcDUT
TYPE ST_Wave42QuantileP10P50P90Output :
STRUCT

	{attribute 'hide'} _header_DO_NOT_CHANGE : ARRAY[0..63] OF SINT := [-1,-112,120,86,52,18,-1,-1,1,-1,0,0,-1,-1,-112,-112,65,64,108,85,118,21,-37,1,110,122,-102,19,93,-117,-35,-43,3,-45,33,-52,25,-24,90,7,83,36,22,5,-43,-65,-103,-61,76,0,0,0,0,0,0,0,0,0,0,0,0,0,0,0];
	out_prediction_tensor : ARRAY[0..0,0..2] OF REAL;

END_STRUCT
END_TYPE

// ---- DUTs/ST_Wave43MixtureDensityK2Input.TcDUT
TYPE ST_Wave43MixtureDensityK2Input :
STRUCT

	{attribute 'hide'} _header_DO_NOT_CHANGE : ARRAY[0..63] OF SINT := [-1,-112,120,86,52,18,-1,-1,1,-1,0,0,-1,-1,-112,-112,55,-22,8,-62,15,-11,-53,-120,-65,-26,40,-59,-103,80,20,5,37,-41,0,-16,-125,-33,-67,117,-59,70,-31,-53,-46,-33,-68,-19,80,2,0,0,0,0,0,0,0,0,0,0,0,0,0,0];
	in_input_tensor : ARRAY[0..0,0..32,0..3] OF REAL;

END_STRUCT
END_TYPE

// ---- DUTs/ST_Wave43MixtureDensityK2Output.TcDUT
TYPE ST_Wave43MixtureDensityK2Output :
STRUCT

	{attribute 'hide'} _header_DO_NOT_CHANGE : ARRAY[0..63] OF SINT := [-1,-112,120,86,52,18,-1,-1,1,-1,0,0,-1,-1,-112,-112,54,-3,-17,51,-108,-42,-47,-97,-51,-21,19,73,46,-30,14,50,-5,-70,67,32,-58,-119,98,-85,10,64,-55,41,100,-21,-124,115,88,0,0,0,0,0,0,0,0,0,0,0,0,0,0,0];
	out_prediction_tensor : ARRAY[0..0,0..5] OF REAL;

END_STRUCT
END_TYPE

// ---- DUTs/ST_Wave43MixtureDensityK3Input.TcDUT
TYPE ST_Wave43MixtureDensityK3Input :
STRUCT

	{attribute 'hide'} _header_DO_NOT_CHANGE : ARRAY[0..63] OF SINT := [-1,-112,120,86,52,18,-1,-1,1,-1,0,0,-1,-1,-112,-112,55,-22,8,-62,15,-11,-53,-120,-65,-26,40,-59,-103,80,20,5,37,-41,0,-16,-125,-33,-67,117,-59,70,-31,-53,-46,-33,-68,-19,80,2,0,0,0,0,0,0,0,0,0,0,0,0,0,0];
	in_input_tensor : ARRAY[0..0,0..32,0..3] OF REAL;

END_STRUCT
END_TYPE

// ---- DUTs/ST_Wave43MixtureDensityK3Output.TcDUT
TYPE ST_Wave43MixtureDensityK3Output :
STRUCT

	{attribute 'hide'} _header_DO_NOT_CHANGE : ARRAY[0..63] OF SINT := [-1,-112,120,86,52,18,-1,-1,1,-1,0,0,-1,-1,-112,-112,-7,125,4,-97,-102,90,119,60,42,56,5,-119,53,39,13,-40,-100,88,-5,50,32,-37,-26,55,-13,-68,-19,-92,59,6,68,-15,100,0,0,0,0,0,0,0,0,0,0,0,0,0,0,0];
	out_prediction_tensor : ARRAY[0..0,0..8] OF REAL;

END_STRUCT
END_TYPE

// ---- DUTs/ST_Wave44CausalTcnLatentOffsetResidualInput.TcDUT
TYPE ST_Wave44CausalTcnLatentOffsetResidualInput :
STRUCT

	{attribute 'hide'} _header_DO_NOT_CHANGE : ARRAY[0..63] OF SINT := [-1,-112,120,86,52,18,-1,-1,1,-1,0,0,-1,-1,-112,-112,55,-22,8,-62,15,-11,-53,-120,-65,-26,40,-59,-103,80,20,5,37,-41,0,-16,-125,-33,-67,117,-59,70,-31,-53,-46,-33,-68,-19,80,2,0,0,0,0,0,0,0,0,0,0,0,0,0,0];
	in_input_tensor : ARRAY[0..0,0..32,0..3] OF REAL;

END_STRUCT
END_TYPE

// ---- DUTs/ST_Wave44CausalTcnLatentOffsetResidualOutput.TcDUT
TYPE ST_Wave44CausalTcnLatentOffsetResidualOutput :
STRUCT

	{attribute 'hide'} _header_DO_NOT_CHANGE : ARRAY[0..63] OF SINT := [-1,-112,120,86,52,18,-1,-1,1,-1,0,0,-1,-1,-112,-112,-35,24,-50,75,-65,96,-121,123,127,87,61,127,-39,-108,16,-70,120,-89,-28,78,-43,26,-32,-7,81,19,29,-89,-55,3,43,2,68,0,0,0,0,0,0,0,0,0,0,0,0,0,0,0];
	out_prediction_tensor : ARRAY[0..0,0..0] OF REAL;

END_STRUCT
END_TYPE

// ---- DUTs/ST_Wave44GruLatentOffsetResidualInput.TcDUT
TYPE ST_Wave44GruLatentOffsetResidualInput :
STRUCT

	{attribute 'hide'} _header_DO_NOT_CHANGE : ARRAY[0..63] OF SINT := [-1,-112,120,86,52,18,-1,-1,1,-1,0,0,-1,-1,-112,-112,55,-22,8,-62,15,-11,-53,-120,-65,-26,40,-59,-103,80,20,5,37,-41,0,-16,-125,-33,-67,117,-59,70,-31,-53,-46,-33,-68,-19,80,2,0,0,0,0,0,0,0,0,0,0,0,0,0,0];
	in_input_tensor : ARRAY[0..0,0..32,0..3] OF REAL;

END_STRUCT
END_TYPE

// ---- DUTs/ST_Wave44GruLatentOffsetResidualOutput.TcDUT
TYPE ST_Wave44GruLatentOffsetResidualOutput :
STRUCT

	{attribute 'hide'} _header_DO_NOT_CHANGE : ARRAY[0..63] OF SINT := [-1,-112,120,86,52,18,-1,-1,1,-1,0,0,-1,-1,-112,-112,-35,24,-50,75,-65,96,-121,123,127,87,61,127,-39,-108,16,-70,120,-89,-28,78,-43,26,-32,-7,81,19,29,-89,-55,3,43,2,68,0,0,0,0,0,0,0,0,0,0,0,0,0,0,0];
	out_prediction_tensor : ARRAY[0..0,0..0] OF REAL;

END_STRUCT
END_TYPE

// ---- DUTs/ST_Wave51HarmonicPriorPointwiseControlInput.TcDUT
TYPE ST_Wave51HarmonicPriorPointwiseControlInput :
STRUCT

	{attribute 'hide'} _header_DO_NOT_CHANGE : ARRAY[0..63] OF SINT := [-1,-112,120,86,52,18,-1,-1,1,-1,0,0,-1,-1,-112,-112,55,-22,8,-62,15,-11,-53,-120,-65,-26,40,-59,-103,80,20,5,37,-41,0,-16,-125,-33,-67,117,-59,70,-31,-53,-46,-33,-68,-19,80,2,0,0,0,0,0,0,0,0,0,0,0,0,0,0];
	in_input_tensor : ARRAY[0..0,0..32,0..3] OF REAL;

END_STRUCT
END_TYPE

// ---- DUTs/ST_Wave51HarmonicPriorPointwiseControlOutput.TcDUT
TYPE ST_Wave51HarmonicPriorPointwiseControlOutput :
STRUCT

	{attribute 'hide'} _header_DO_NOT_CHANGE : ARRAY[0..63] OF SINT := [-1,-112,120,86,52,18,-1,-1,1,-1,0,0,-1,-1,-112,-112,-35,24,-50,75,-65,96,-121,123,127,87,61,127,-39,-108,16,-70,120,-89,-28,78,-43,26,-32,-7,81,19,29,-89,-55,3,43,2,68,0,0,0,0,0,0,0,0,0,0,0,0,0,0,0];
	out_prediction_tensor : ARRAY[0..0,0..0] OF REAL;

END_STRUCT
END_TYPE

// ---- DUTs/ST_Wave51HarmonicPriorSmoothL1StructuredInput.TcDUT
TYPE ST_Wave51HarmonicPriorSmoothL1StructuredInput :
STRUCT

	{attribute 'hide'} _header_DO_NOT_CHANGE : ARRAY[0..63] OF SINT := [-1,-112,120,86,52,18,-1,-1,1,-1,0,0,-1,-1,-112,-112,55,-22,8,-62,15,-11,-53,-120,-65,-26,40,-59,-103,80,20,5,37,-41,0,-16,-125,-33,-67,117,-59,70,-31,-53,-46,-33,-68,-19,80,2,0,0,0,0,0,0,0,0,0,0,0,0,0,0];
	in_input_tensor : ARRAY[0..0,0..32,0..3] OF REAL;

END_STRUCT
END_TYPE

// ---- DUTs/ST_Wave51HarmonicPriorSmoothL1StructuredOutput.TcDUT
TYPE ST_Wave51HarmonicPriorSmoothL1StructuredOutput :
STRUCT

	{attribute 'hide'} _header_DO_NOT_CHANGE : ARRAY[0..63] OF SINT := [-1,-112,120,86,52,18,-1,-1,1,-1,0,0,-1,-1,-112,-112,-35,24,-50,75,-65,96,-121,123,127,87,61,127,-39,-108,16,-70,120,-89,-28,78,-43,26,-32,-7,81,19,29,-89,-55,3,43,2,68,0,0,0,0,0,0,0,0,0,0,0,0,0,0,0];
	out_prediction_tensor : ARRAY[0..0,0..0] OF REAL;

END_STRUCT
END_TYPE

// ---- POUs/P_TF3820StandaloneModelTest.TcPOU
PROGRAM P_TF3820StandaloneModelTest
VAR_INPUT
	SelectedModel		: E_TF3820StandaloneModelId := E_TF3820StandaloneModelId.Model_Feedforward;
	bLoadSelectedModel	: BOOL := TRUE;
	bEnablePrediction	: BOOL := TRUE;
	bReset				: BOOL;
	sMlSvrNetId			: T_MaxString := 'local';
	eExecutionProvider	: E_ExecutionProvider := E_ExecutionProvider.CPU;
	nConfigureTimeout	: UDINT := 1000;
	nPredictTimeout		: UDINT := 100;
	nPriority			: UDINT := 0;
	fTheta					: REAL := 0.0;
	fThetaDot				: REAL := 500.0;
	fTorque				: REAL := 100.0;
	fTemperature			: REAL := 30.0;
	fDirectionFlag		: REAL := 1.0;
	fThetaStep			: REAL := 0.25;
END_VAR
VAR_OUTPUT
	bConfigured			: BOOL;
	bBusy					: BOOL;
	bPredictionPending	: BOOL;
	bPredictionReady	: BOOL;
	bResetDone			: BOOL;
	bError					: BOOL;
	nErrorCode			: HRESULT;
	nMaxInferenceDuration	: UDINT;
	aPredictionOutput	: ARRAY[0..8] OF REAL;
END_VAR
VAR
	fbFeedforward	: FB_FeedforwardTf3820Runner;
	fbGruSequence	: FB_GruSequenceTf3820Runner;
	fbHarmonicRegression	: FB_HarmonicRegressionTf3820Runner;
	fbLstmSequence	: FB_LstmSequenceTf3820Runner;
	fbPeriodicGruSequence	: FB_PeriodicGruSequenceTf3820Runner;
	fbPeriodicLstmSequence	: FB_PeriodicLstmSequenceTf3820Runner;
	fbPeriodicMlp	: FB_PeriodicMlpTf3820Runner;
	fbPeriodicMlpHarmonic	: FB_PeriodicMlpHarmonicTf3820Runner;
	fbPeriodicTemporalConvolution	: FB_PeriodicTemporalConvolutionTf3820Runner;
	fbRcimTrack1	: FB_RcimTrack1Tf3820Runner;
	fbResidualHarmonicGruSequenceDense240	: FB_ResidualHarmonicGruSequenceDense240Tf3820Runner;
	fbResidualHarmonicGruSequenceDense360	: FB_ResidualHarmonicGruSequenceDense360Tf3820Runner;
	fbResidualHarmonicGruSequenceSparseRcim	: FB_ResidualHarmonicGruSequenceSparseRcimTf3820Runner;
	fbResidualHarmonicLstmSequenceDense240	: FB_ResidualHarmonicLstmSequenceDense240Tf3820Runner;
	fbResidualHarmonicLstmSequenceDense360	: FB_ResidualHarmonicLstmSequenceDense360Tf3820Runner;
	fbResidualHarmonicLstmSequenceSparseRcim	: FB_ResidualHarmonicLstmSequenceSparseRcimTf3820Runner;
	fbResidualHarmonicMlp	: FB_ResidualHarmonicMlpTf3820Runner;
	fbTemporalConvolution	: FB_TemporalConvolutionTf3820Runner;
	fbTree	: FB_TreeTf3820Runner;
	fbWave31SequentialResidualOffsetProbe	: FB_Wave31SequentialResidualOffsetProbeTf3820Runner;
	fbWave32CleanSequentialResidualOffset	: FB_Wave32CleanSequentialResidualOffsetTf3820Runner;
	fbWave32HarmonicResidualOffset	: FB_Wave32HarmonicResidualOffsetTf3820Runner;
	fbWave33CurveAwarePointwiseControl	: FB_Wave33CurveAwarePointwiseControlTf3820Runner;
	fbWave33FullCurveComposite	: FB_Wave33FullCurveCompositeTf3820Runner;
	fbWave33RawCenteredShapeCurveAware	: FB_Wave33RawCenteredShapeCurveAwareTf3820Runner;
	fbWave33RawOffsetCurveAware	: FB_Wave33RawOffsetCurveAwareTf3820Runner;
	fbWave41LogCoshRobustLoss	: FB_Wave41LogCoshRobustLossTf3820Runner;
	fbWave41MaeRobustLoss	: FB_Wave41MaeRobustLossTf3820Runner;
	fbWave41SmoothL1RobustLoss	: FB_Wave41SmoothL1RobustLossTf3820Runner;
	fbWave42GaussianNll	: FB_Wave42GaussianNllTf3820Runner;
	fbWave42QuantileP10P50P90	: FB_Wave42QuantileP10P50P90Tf3820Runner;
	fbWave43MixtureDensityK2	: FB_Wave43MixtureDensityK2Tf3820Runner;
	fbWave43MixtureDensityK3	: FB_Wave43MixtureDensityK3Tf3820Runner;
	fbWave44CausalTcnLatentOffsetResidual	: FB_Wave44CausalTcnLatentOffsetResidualTf3820Runner;
	fbWave44GruLatentOffsetResidual	: FB_Wave44GruLatentOffsetResidualTf3820Runner;
	fbWave51HarmonicPriorPointwiseControl	: FB_Wave51HarmonicPriorPointwiseControlTf3820Runner;
	fbWave51HarmonicPriorSmoothL1Structured	: FB_Wave51HarmonicPriorSmoothL1StructuredTf3820Runner;
END_VAR

CASE SelectedModel OF
	E_TF3820StandaloneModelId.Model_Feedforward:
		fbFeedforward(
			sModelJsonFilePath := 'C:\TwinCAT\3.1\Boot\ML\tf3820\standalone\feedforward\model.json',
			sMlSvrNetId := sMlSvrNetId,
			eExecutionProvider := eExecutionProvider,
			bEnable := bEnablePrediction,
			bReset := bReset,
			bLoadModel := bLoadSelectedModel,
			nConfigureTimeout := nConfigureTimeout,
			nPredictTimeout := nPredictTimeout,
			nPriority := nPriority,
			fTheta := fTheta,
			fThetaDot := fThetaDot,
			fTorque := fTorque,
			fTemperature := fTemperature,
			fDirectionFlag := fDirectionFlag,
			fThetaStep := fThetaStep,
			bConfigured => bConfigured,
			bBusy => bBusy,
			bPredictionPending => bPredictionPending,
			bPredictionReady => bPredictionReady,
			bResetDone => bResetDone,
			bError => bError,
			nErrorCode => nErrorCode,
			nMaxInferenceDuration => nMaxInferenceDuration,
			aPredictionOutput => aPredictionOutput);
	E_TF3820StandaloneModelId.Model_Gru_Sequence:
		fbGruSequence(
			sModelJsonFilePath := 'C:\TwinCAT\3.1\Boot\ML\tf3820\standalone\gru_sequence\model.json',
			sMlSvrNetId := sMlSvrNetId,
			eExecutionProvider := eExecutionProvider,
			bEnable := bEnablePrediction,
			bReset := bReset,
			bLoadModel := bLoadSelectedModel,
			nConfigureTimeout := nConfigureTimeout,
			nPredictTimeout := nPredictTimeout,
			nPriority := nPriority,
			fTheta := fTheta,
			fThetaDot := fThetaDot,
			fTorque := fTorque,
			fTemperature := fTemperature,
			fDirectionFlag := fDirectionFlag,
			fThetaStep := fThetaStep,
			bConfigured => bConfigured,
			bBusy => bBusy,
			bPredictionPending => bPredictionPending,
			bPredictionReady => bPredictionReady,
			bResetDone => bResetDone,
			bError => bError,
			nErrorCode => nErrorCode,
			nMaxInferenceDuration => nMaxInferenceDuration,
			aPredictionOutput => aPredictionOutput);
	E_TF3820StandaloneModelId.Model_Harmonic_Regression:
		fbHarmonicRegression(
			sModelJsonFilePath := 'C:\TwinCAT\3.1\Boot\ML\tf3820\standalone\harmonic_regression\model.json',
			sMlSvrNetId := sMlSvrNetId,
			eExecutionProvider := eExecutionProvider,
			bEnable := bEnablePrediction,
			bReset := bReset,
			bLoadModel := bLoadSelectedModel,
			nConfigureTimeout := nConfigureTimeout,
			nPredictTimeout := nPredictTimeout,
			nPriority := nPriority,
			fTheta := fTheta,
			fThetaDot := fThetaDot,
			fTorque := fTorque,
			fTemperature := fTemperature,
			fDirectionFlag := fDirectionFlag,
			fThetaStep := fThetaStep,
			bConfigured => bConfigured,
			bBusy => bBusy,
			bPredictionPending => bPredictionPending,
			bPredictionReady => bPredictionReady,
			bResetDone => bResetDone,
			bError => bError,
			nErrorCode => nErrorCode,
			nMaxInferenceDuration => nMaxInferenceDuration,
			aPredictionOutput => aPredictionOutput);
	E_TF3820StandaloneModelId.Model_Lstm_Sequence:
		fbLstmSequence(
			sModelJsonFilePath := 'C:\TwinCAT\3.1\Boot\ML\tf3820\standalone\lstm_sequence\model.json',
			sMlSvrNetId := sMlSvrNetId,
			eExecutionProvider := eExecutionProvider,
			bEnable := bEnablePrediction,
			bReset := bReset,
			bLoadModel := bLoadSelectedModel,
			nConfigureTimeout := nConfigureTimeout,
			nPredictTimeout := nPredictTimeout,
			nPriority := nPriority,
			fTheta := fTheta,
			fThetaDot := fThetaDot,
			fTorque := fTorque,
			fTemperature := fTemperature,
			fDirectionFlag := fDirectionFlag,
			fThetaStep := fThetaStep,
			bConfigured => bConfigured,
			bBusy => bBusy,
			bPredictionPending => bPredictionPending,
			bPredictionReady => bPredictionReady,
			bResetDone => bResetDone,
			bError => bError,
			nErrorCode => nErrorCode,
			nMaxInferenceDuration => nMaxInferenceDuration,
			aPredictionOutput => aPredictionOutput);
	E_TF3820StandaloneModelId.Model_Periodic_Gru_Sequence:
		fbPeriodicGruSequence(
			sModelJsonFilePath := 'C:\TwinCAT\3.1\Boot\ML\tf3820\standalone\periodic_gru_sequence\model.json',
			sMlSvrNetId := sMlSvrNetId,
			eExecutionProvider := eExecutionProvider,
			bEnable := bEnablePrediction,
			bReset := bReset,
			bLoadModel := bLoadSelectedModel,
			nConfigureTimeout := nConfigureTimeout,
			nPredictTimeout := nPredictTimeout,
			nPriority := nPriority,
			fTheta := fTheta,
			fThetaDot := fThetaDot,
			fTorque := fTorque,
			fTemperature := fTemperature,
			fDirectionFlag := fDirectionFlag,
			fThetaStep := fThetaStep,
			bConfigured => bConfigured,
			bBusy => bBusy,
			bPredictionPending => bPredictionPending,
			bPredictionReady => bPredictionReady,
			bResetDone => bResetDone,
			bError => bError,
			nErrorCode => nErrorCode,
			nMaxInferenceDuration => nMaxInferenceDuration,
			aPredictionOutput => aPredictionOutput);
	E_TF3820StandaloneModelId.Model_Periodic_Lstm_Sequence:
		fbPeriodicLstmSequence(
			sModelJsonFilePath := 'C:\TwinCAT\3.1\Boot\ML\tf3820\standalone\periodic_lstm_sequence\model.json',
			sMlSvrNetId := sMlSvrNetId,
			eExecutionProvider := eExecutionProvider,
			bEnable := bEnablePrediction,
			bReset := bReset,
			bLoadModel := bLoadSelectedModel,
			nConfigureTimeout := nConfigureTimeout,
			nPredictTimeout := nPredictTimeout,
			nPriority := nPriority,
			fTheta := fTheta,
			fThetaDot := fThetaDot,
			fTorque := fTorque,
			fTemperature := fTemperature,
			fDirectionFlag := fDirectionFlag,
			fThetaStep := fThetaStep,
			bConfigured => bConfigured,
			bBusy => bBusy,
			bPredictionPending => bPredictionPending,
			bPredictionReady => bPredictionReady,
			bResetDone => bResetDone,
			bError => bError,
			nErrorCode => nErrorCode,
			nMaxInferenceDuration => nMaxInferenceDuration,
			aPredictionOutput => aPredictionOutput);
	E_TF3820StandaloneModelId.Model_Periodic_Mlp:
		fbPeriodicMlp(
			sModelJsonFilePath := 'C:\TwinCAT\3.1\Boot\ML\tf3820\standalone\periodic_mlp\model.json',
			sMlSvrNetId := sMlSvrNetId,
			eExecutionProvider := eExecutionProvider,
			bEnable := bEnablePrediction,
			bReset := bReset,
			bLoadModel := bLoadSelectedModel,
			nConfigureTimeout := nConfigureTimeout,
			nPredictTimeout := nPredictTimeout,
			nPriority := nPriority,
			fTheta := fTheta,
			fThetaDot := fThetaDot,
			fTorque := fTorque,
			fTemperature := fTemperature,
			fDirectionFlag := fDirectionFlag,
			fThetaStep := fThetaStep,
			bConfigured => bConfigured,
			bBusy => bBusy,
			bPredictionPending => bPredictionPending,
			bPredictionReady => bPredictionReady,
			bResetDone => bResetDone,
			bError => bError,
			nErrorCode => nErrorCode,
			nMaxInferenceDuration => nMaxInferenceDuration,
			aPredictionOutput => aPredictionOutput);
	E_TF3820StandaloneModelId.Model_Periodic_Mlp_Harmonic:
		fbPeriodicMlpHarmonic(
			sModelJsonFilePath := 'C:\TwinCAT\3.1\Boot\ML\tf3820\standalone\periodic_mlp_harmonic\model.json',
			sMlSvrNetId := sMlSvrNetId,
			eExecutionProvider := eExecutionProvider,
			bEnable := bEnablePrediction,
			bReset := bReset,
			bLoadModel := bLoadSelectedModel,
			nConfigureTimeout := nConfigureTimeout,
			nPredictTimeout := nPredictTimeout,
			nPriority := nPriority,
			fTheta := fTheta,
			fThetaDot := fThetaDot,
			fTorque := fTorque,
			fTemperature := fTemperature,
			fDirectionFlag := fDirectionFlag,
			fThetaStep := fThetaStep,
			bConfigured => bConfigured,
			bBusy => bBusy,
			bPredictionPending => bPredictionPending,
			bPredictionReady => bPredictionReady,
			bResetDone => bResetDone,
			bError => bError,
			nErrorCode => nErrorCode,
			nMaxInferenceDuration => nMaxInferenceDuration,
			aPredictionOutput => aPredictionOutput);
	E_TF3820StandaloneModelId.Model_Periodic_Temporal_Convolution:
		fbPeriodicTemporalConvolution(
			sModelJsonFilePath := 'C:\TwinCAT\3.1\Boot\ML\tf3820\standalone\periodic_temporal_convolution\model.json',
			sMlSvrNetId := sMlSvrNetId,
			eExecutionProvider := eExecutionProvider,
			bEnable := bEnablePrediction,
			bReset := bReset,
			bLoadModel := bLoadSelectedModel,
			nConfigureTimeout := nConfigureTimeout,
			nPredictTimeout := nPredictTimeout,
			nPriority := nPriority,
			fTheta := fTheta,
			fThetaDot := fThetaDot,
			fTorque := fTorque,
			fTemperature := fTemperature,
			fDirectionFlag := fDirectionFlag,
			fThetaStep := fThetaStep,
			bConfigured => bConfigured,
			bBusy => bBusy,
			bPredictionPending => bPredictionPending,
			bPredictionReady => bPredictionReady,
			bResetDone => bResetDone,
			bError => bError,
			nErrorCode => nErrorCode,
			nMaxInferenceDuration => nMaxInferenceDuration,
			aPredictionOutput => aPredictionOutput);
	E_TF3820StandaloneModelId.Model_Rcim_Track1:
		fbRcimTrack1(
			sModelJsonFilePath := 'C:\TwinCAT\3.1\Boot\ML\tf3820\standalone\rcim_track1\model.json',
			sMlSvrNetId := sMlSvrNetId,
			eExecutionProvider := eExecutionProvider,
			bEnable := bEnablePrediction,
			bReset := bReset,
			bLoadModel := bLoadSelectedModel,
			nConfigureTimeout := nConfigureTimeout,
			nPredictTimeout := nPredictTimeout,
			nPriority := nPriority,
			fTheta := fTheta,
			fThetaDot := fThetaDot,
			fTorque := fTorque,
			fTemperature := fTemperature,
			fDirectionFlag := fDirectionFlag,
			fThetaStep := fThetaStep,
			bConfigured => bConfigured,
			bBusy => bBusy,
			bPredictionPending => bPredictionPending,
			bPredictionReady => bPredictionReady,
			bResetDone => bResetDone,
			bError => bError,
			nErrorCode => nErrorCode,
			nMaxInferenceDuration => nMaxInferenceDuration,
			aPredictionOutput => aPredictionOutput);
	E_TF3820StandaloneModelId.Model_Residual_Harmonic_Gru_Sequence_Dense240:
		fbResidualHarmonicGruSequenceDense240(
			sModelJsonFilePath := 'C:\TwinCAT\3.1\Boot\ML\tf3820\standalone\residual_harmonic_gru_sequence_dense240\model.json',
			sMlSvrNetId := sMlSvrNetId,
			eExecutionProvider := eExecutionProvider,
			bEnable := bEnablePrediction,
			bReset := bReset,
			bLoadModel := bLoadSelectedModel,
			nConfigureTimeout := nConfigureTimeout,
			nPredictTimeout := nPredictTimeout,
			nPriority := nPriority,
			fTheta := fTheta,
			fThetaDot := fThetaDot,
			fTorque := fTorque,
			fTemperature := fTemperature,
			fDirectionFlag := fDirectionFlag,
			fThetaStep := fThetaStep,
			bConfigured => bConfigured,
			bBusy => bBusy,
			bPredictionPending => bPredictionPending,
			bPredictionReady => bPredictionReady,
			bResetDone => bResetDone,
			bError => bError,
			nErrorCode => nErrorCode,
			nMaxInferenceDuration => nMaxInferenceDuration,
			aPredictionOutput => aPredictionOutput);
	E_TF3820StandaloneModelId.Model_Residual_Harmonic_Gru_Sequence_Dense360:
		fbResidualHarmonicGruSequenceDense360(
			sModelJsonFilePath := 'C:\TwinCAT\3.1\Boot\ML\tf3820\standalone\residual_harmonic_gru_sequence_dense360\model.json',
			sMlSvrNetId := sMlSvrNetId,
			eExecutionProvider := eExecutionProvider,
			bEnable := bEnablePrediction,
			bReset := bReset,
			bLoadModel := bLoadSelectedModel,
			nConfigureTimeout := nConfigureTimeout,
			nPredictTimeout := nPredictTimeout,
			nPriority := nPriority,
			fTheta := fTheta,
			fThetaDot := fThetaDot,
			fTorque := fTorque,
			fTemperature := fTemperature,
			fDirectionFlag := fDirectionFlag,
			fThetaStep := fThetaStep,
			bConfigured => bConfigured,
			bBusy => bBusy,
			bPredictionPending => bPredictionPending,
			bPredictionReady => bPredictionReady,
			bResetDone => bResetDone,
			bError => bError,
			nErrorCode => nErrorCode,
			nMaxInferenceDuration => nMaxInferenceDuration,
			aPredictionOutput => aPredictionOutput);
	E_TF3820StandaloneModelId.Model_Residual_Harmonic_Gru_Sequence_Sparse_Rcim:
		fbResidualHarmonicGruSequenceSparseRcim(
			sModelJsonFilePath := 'C:\TwinCAT\3.1\Boot\ML\tf3820\standalone\residual_harmonic_gru_sequence_sparse_rcim\model.json',
			sMlSvrNetId := sMlSvrNetId,
			eExecutionProvider := eExecutionProvider,
			bEnable := bEnablePrediction,
			bReset := bReset,
			bLoadModel := bLoadSelectedModel,
			nConfigureTimeout := nConfigureTimeout,
			nPredictTimeout := nPredictTimeout,
			nPriority := nPriority,
			fTheta := fTheta,
			fThetaDot := fThetaDot,
			fTorque := fTorque,
			fTemperature := fTemperature,
			fDirectionFlag := fDirectionFlag,
			fThetaStep := fThetaStep,
			bConfigured => bConfigured,
			bBusy => bBusy,
			bPredictionPending => bPredictionPending,
			bPredictionReady => bPredictionReady,
			bResetDone => bResetDone,
			bError => bError,
			nErrorCode => nErrorCode,
			nMaxInferenceDuration => nMaxInferenceDuration,
			aPredictionOutput => aPredictionOutput);
	E_TF3820StandaloneModelId.Model_Residual_Harmonic_Lstm_Sequence_Dense240:
		fbResidualHarmonicLstmSequenceDense240(
			sModelJsonFilePath := 'C:\TwinCAT\3.1\Boot\ML\tf3820\standalone\residual_harmonic_lstm_sequence_dense240\model.json',
			sMlSvrNetId := sMlSvrNetId,
			eExecutionProvider := eExecutionProvider,
			bEnable := bEnablePrediction,
			bReset := bReset,
			bLoadModel := bLoadSelectedModel,
			nConfigureTimeout := nConfigureTimeout,
			nPredictTimeout := nPredictTimeout,
			nPriority := nPriority,
			fTheta := fTheta,
			fThetaDot := fThetaDot,
			fTorque := fTorque,
			fTemperature := fTemperature,
			fDirectionFlag := fDirectionFlag,
			fThetaStep := fThetaStep,
			bConfigured => bConfigured,
			bBusy => bBusy,
			bPredictionPending => bPredictionPending,
			bPredictionReady => bPredictionReady,
			bResetDone => bResetDone,
			bError => bError,
			nErrorCode => nErrorCode,
			nMaxInferenceDuration => nMaxInferenceDuration,
			aPredictionOutput => aPredictionOutput);
	E_TF3820StandaloneModelId.Model_Residual_Harmonic_Lstm_Sequence_Dense360:
		fbResidualHarmonicLstmSequenceDense360(
			sModelJsonFilePath := 'C:\TwinCAT\3.1\Boot\ML\tf3820\standalone\residual_harmonic_lstm_sequence_dense360\model.json',
			sMlSvrNetId := sMlSvrNetId,
			eExecutionProvider := eExecutionProvider,
			bEnable := bEnablePrediction,
			bReset := bReset,
			bLoadModel := bLoadSelectedModel,
			nConfigureTimeout := nConfigureTimeout,
			nPredictTimeout := nPredictTimeout,
			nPriority := nPriority,
			fTheta := fTheta,
			fThetaDot := fThetaDot,
			fTorque := fTorque,
			fTemperature := fTemperature,
			fDirectionFlag := fDirectionFlag,
			fThetaStep := fThetaStep,
			bConfigured => bConfigured,
			bBusy => bBusy,
			bPredictionPending => bPredictionPending,
			bPredictionReady => bPredictionReady,
			bResetDone => bResetDone,
			bError => bError,
			nErrorCode => nErrorCode,
			nMaxInferenceDuration => nMaxInferenceDuration,
			aPredictionOutput => aPredictionOutput);
	E_TF3820StandaloneModelId.Model_Residual_Harmonic_Lstm_Sequence_Sparse_Rcim:
		fbResidualHarmonicLstmSequenceSparseRcim(
			sModelJsonFilePath := 'C:\TwinCAT\3.1\Boot\ML\tf3820\standalone\residual_harmonic_lstm_sequence_sparse_rcim\model.json',
			sMlSvrNetId := sMlSvrNetId,
			eExecutionProvider := eExecutionProvider,
			bEnable := bEnablePrediction,
			bReset := bReset,
			bLoadModel := bLoadSelectedModel,
			nConfigureTimeout := nConfigureTimeout,
			nPredictTimeout := nPredictTimeout,
			nPriority := nPriority,
			fTheta := fTheta,
			fThetaDot := fThetaDot,
			fTorque := fTorque,
			fTemperature := fTemperature,
			fDirectionFlag := fDirectionFlag,
			fThetaStep := fThetaStep,
			bConfigured => bConfigured,
			bBusy => bBusy,
			bPredictionPending => bPredictionPending,
			bPredictionReady => bPredictionReady,
			bResetDone => bResetDone,
			bError => bError,
			nErrorCode => nErrorCode,
			nMaxInferenceDuration => nMaxInferenceDuration,
			aPredictionOutput => aPredictionOutput);
	E_TF3820StandaloneModelId.Model_Residual_Harmonic_Mlp:
		fbResidualHarmonicMlp(
			sModelJsonFilePath := 'C:\TwinCAT\3.1\Boot\ML\tf3820\standalone\residual_harmonic_mlp\model.json',
			sMlSvrNetId := sMlSvrNetId,
			eExecutionProvider := eExecutionProvider,
			bEnable := bEnablePrediction,
			bReset := bReset,
			bLoadModel := bLoadSelectedModel,
			nConfigureTimeout := nConfigureTimeout,
			nPredictTimeout := nPredictTimeout,
			nPriority := nPriority,
			fTheta := fTheta,
			fThetaDot := fThetaDot,
			fTorque := fTorque,
			fTemperature := fTemperature,
			fDirectionFlag := fDirectionFlag,
			fThetaStep := fThetaStep,
			bConfigured => bConfigured,
			bBusy => bBusy,
			bPredictionPending => bPredictionPending,
			bPredictionReady => bPredictionReady,
			bResetDone => bResetDone,
			bError => bError,
			nErrorCode => nErrorCode,
			nMaxInferenceDuration => nMaxInferenceDuration,
			aPredictionOutput => aPredictionOutput);
	E_TF3820StandaloneModelId.Model_Temporal_Convolution:
		fbTemporalConvolution(
			sModelJsonFilePath := 'C:\TwinCAT\3.1\Boot\ML\tf3820\standalone\temporal_convolution\model.json',
			sMlSvrNetId := sMlSvrNetId,
			eExecutionProvider := eExecutionProvider,
			bEnable := bEnablePrediction,
			bReset := bReset,
			bLoadModel := bLoadSelectedModel,
			nConfigureTimeout := nConfigureTimeout,
			nPredictTimeout := nPredictTimeout,
			nPriority := nPriority,
			fTheta := fTheta,
			fThetaDot := fThetaDot,
			fTorque := fTorque,
			fTemperature := fTemperature,
			fDirectionFlag := fDirectionFlag,
			fThetaStep := fThetaStep,
			bConfigured => bConfigured,
			bBusy => bBusy,
			bPredictionPending => bPredictionPending,
			bPredictionReady => bPredictionReady,
			bResetDone => bResetDone,
			bError => bError,
			nErrorCode => nErrorCode,
			nMaxInferenceDuration => nMaxInferenceDuration,
			aPredictionOutput => aPredictionOutput);
	E_TF3820StandaloneModelId.Model_Tree:
		fbTree(
			sModelJsonFilePath := 'C:\TwinCAT\3.1\Boot\ML\tf3820\standalone\tree\model.json',
			sMlSvrNetId := sMlSvrNetId,
			eExecutionProvider := eExecutionProvider,
			bEnable := bEnablePrediction,
			bReset := bReset,
			bLoadModel := bLoadSelectedModel,
			nConfigureTimeout := nConfigureTimeout,
			nPredictTimeout := nPredictTimeout,
			nPriority := nPriority,
			fTheta := fTheta,
			fThetaDot := fThetaDot,
			fTorque := fTorque,
			fTemperature := fTemperature,
			fDirectionFlag := fDirectionFlag,
			fThetaStep := fThetaStep,
			bConfigured => bConfigured,
			bBusy => bBusy,
			bPredictionPending => bPredictionPending,
			bPredictionReady => bPredictionReady,
			bResetDone => bResetDone,
			bError => bError,
			nErrorCode => nErrorCode,
			nMaxInferenceDuration => nMaxInferenceDuration,
			aPredictionOutput => aPredictionOutput);
	E_TF3820StandaloneModelId.Model_Wave3_1_Sequential_Residual_Offset_Probe:
		fbWave31SequentialResidualOffsetProbe(
			sModelJsonFilePath := 'C:\TwinCAT\3.1\Boot\ML\tf3820\standalone\wave3_1_sequential_residual_offset_probe\model.json',
			sMlSvrNetId := sMlSvrNetId,
			eExecutionProvider := eExecutionProvider,
			bEnable := bEnablePrediction,
			bReset := bReset,
			bLoadModel := bLoadSelectedModel,
			nConfigureTimeout := nConfigureTimeout,
			nPredictTimeout := nPredictTimeout,
			nPriority := nPriority,
			fTheta := fTheta,
			fThetaDot := fThetaDot,
			fTorque := fTorque,
			fTemperature := fTemperature,
			fDirectionFlag := fDirectionFlag,
			fThetaStep := fThetaStep,
			bConfigured => bConfigured,
			bBusy => bBusy,
			bPredictionPending => bPredictionPending,
			bPredictionReady => bPredictionReady,
			bResetDone => bResetDone,
			bError => bError,
			nErrorCode => nErrorCode,
			nMaxInferenceDuration => nMaxInferenceDuration,
			aPredictionOutput => aPredictionOutput);
	E_TF3820StandaloneModelId.Model_Wave3_2_Clean_Sequential_Residual_Offset:
		fbWave32CleanSequentialResidualOffset(
			sModelJsonFilePath := 'C:\TwinCAT\3.1\Boot\ML\tf3820\standalone\wave3_2_clean_sequential_residual_offset\model.json',
			sMlSvrNetId := sMlSvrNetId,
			eExecutionProvider := eExecutionProvider,
			bEnable := bEnablePrediction,
			bReset := bReset,
			bLoadModel := bLoadSelectedModel,
			nConfigureTimeout := nConfigureTimeout,
			nPredictTimeout := nPredictTimeout,
			nPriority := nPriority,
			fTheta := fTheta,
			fThetaDot := fThetaDot,
			fTorque := fTorque,
			fTemperature := fTemperature,
			fDirectionFlag := fDirectionFlag,
			fThetaStep := fThetaStep,
			bConfigured => bConfigured,
			bBusy => bBusy,
			bPredictionPending => bPredictionPending,
			bPredictionReady => bPredictionReady,
			bResetDone => bResetDone,
			bError => bError,
			nErrorCode => nErrorCode,
			nMaxInferenceDuration => nMaxInferenceDuration,
			aPredictionOutput => aPredictionOutput);
	E_TF3820StandaloneModelId.Model_Wave3_2_Harmonic_Residual_Offset:
		fbWave32HarmonicResidualOffset(
			sModelJsonFilePath := 'C:\TwinCAT\3.1\Boot\ML\tf3820\standalone\wave3_2_harmonic_residual_offset\model.json',
			sMlSvrNetId := sMlSvrNetId,
			eExecutionProvider := eExecutionProvider,
			bEnable := bEnablePrediction,
			bReset := bReset,
			bLoadModel := bLoadSelectedModel,
			nConfigureTimeout := nConfigureTimeout,
			nPredictTimeout := nPredictTimeout,
			nPriority := nPriority,
			fTheta := fTheta,
			fThetaDot := fThetaDot,
			fTorque := fTorque,
			fTemperature := fTemperature,
			fDirectionFlag := fDirectionFlag,
			fThetaStep := fThetaStep,
			bConfigured => bConfigured,
			bBusy => bBusy,
			bPredictionPending => bPredictionPending,
			bPredictionReady => bPredictionReady,
			bResetDone => bResetDone,
			bError => bError,
			nErrorCode => nErrorCode,
			nMaxInferenceDuration => nMaxInferenceDuration,
			aPredictionOutput => aPredictionOutput);
	E_TF3820StandaloneModelId.Model_Wave3_3_Curve_Aware_Pointwise_Control:
		fbWave33CurveAwarePointwiseControl(
			sModelJsonFilePath := 'C:\TwinCAT\3.1\Boot\ML\tf3820\standalone\wave3_3_curve_aware_pointwise_control\model.json',
			sMlSvrNetId := sMlSvrNetId,
			eExecutionProvider := eExecutionProvider,
			bEnable := bEnablePrediction,
			bReset := bReset,
			bLoadModel := bLoadSelectedModel,
			nConfigureTimeout := nConfigureTimeout,
			nPredictTimeout := nPredictTimeout,
			nPriority := nPriority,
			fTheta := fTheta,
			fThetaDot := fThetaDot,
			fTorque := fTorque,
			fTemperature := fTemperature,
			fDirectionFlag := fDirectionFlag,
			fThetaStep := fThetaStep,
			bConfigured => bConfigured,
			bBusy => bBusy,
			bPredictionPending => bPredictionPending,
			bPredictionReady => bPredictionReady,
			bResetDone => bResetDone,
			bError => bError,
			nErrorCode => nErrorCode,
			nMaxInferenceDuration => nMaxInferenceDuration,
			aPredictionOutput => aPredictionOutput);
	E_TF3820StandaloneModelId.Model_Wave3_3_Full_Curve_Composite:
		fbWave33FullCurveComposite(
			sModelJsonFilePath := 'C:\TwinCAT\3.1\Boot\ML\tf3820\standalone\wave3_3_full_curve_composite\model.json',
			sMlSvrNetId := sMlSvrNetId,
			eExecutionProvider := eExecutionProvider,
			bEnable := bEnablePrediction,
			bReset := bReset,
			bLoadModel := bLoadSelectedModel,
			nConfigureTimeout := nConfigureTimeout,
			nPredictTimeout := nPredictTimeout,
			nPriority := nPriority,
			fTheta := fTheta,
			fThetaDot := fThetaDot,
			fTorque := fTorque,
			fTemperature := fTemperature,
			fDirectionFlag := fDirectionFlag,
			fThetaStep := fThetaStep,
			bConfigured => bConfigured,
			bBusy => bBusy,
			bPredictionPending => bPredictionPending,
			bPredictionReady => bPredictionReady,
			bResetDone => bResetDone,
			bError => bError,
			nErrorCode => nErrorCode,
			nMaxInferenceDuration => nMaxInferenceDuration,
			aPredictionOutput => aPredictionOutput);
	E_TF3820StandaloneModelId.Model_Wave3_3_Raw_Centered_Shape_Curve_Aware:
		fbWave33RawCenteredShapeCurveAware(
			sModelJsonFilePath := 'C:\TwinCAT\3.1\Boot\ML\tf3820\standalone\wave3_3_raw_centered_shape_curve_aware\model.json',
			sMlSvrNetId := sMlSvrNetId,
			eExecutionProvider := eExecutionProvider,
			bEnable := bEnablePrediction,
			bReset := bReset,
			bLoadModel := bLoadSelectedModel,
			nConfigureTimeout := nConfigureTimeout,
			nPredictTimeout := nPredictTimeout,
			nPriority := nPriority,
			fTheta := fTheta,
			fThetaDot := fThetaDot,
			fTorque := fTorque,
			fTemperature := fTemperature,
			fDirectionFlag := fDirectionFlag,
			fThetaStep := fThetaStep,
			bConfigured => bConfigured,
			bBusy => bBusy,
			bPredictionPending => bPredictionPending,
			bPredictionReady => bPredictionReady,
			bResetDone => bResetDone,
			bError => bError,
			nErrorCode => nErrorCode,
			nMaxInferenceDuration => nMaxInferenceDuration,
			aPredictionOutput => aPredictionOutput);
	E_TF3820StandaloneModelId.Model_Wave3_3_Raw_Offset_Curve_Aware:
		fbWave33RawOffsetCurveAware(
			sModelJsonFilePath := 'C:\TwinCAT\3.1\Boot\ML\tf3820\standalone\wave3_3_raw_offset_curve_aware\model.json',
			sMlSvrNetId := sMlSvrNetId,
			eExecutionProvider := eExecutionProvider,
			bEnable := bEnablePrediction,
			bReset := bReset,
			bLoadModel := bLoadSelectedModel,
			nConfigureTimeout := nConfigureTimeout,
			nPredictTimeout := nPredictTimeout,
			nPriority := nPriority,
			fTheta := fTheta,
			fThetaDot := fThetaDot,
			fTorque := fTorque,
			fTemperature := fTemperature,
			fDirectionFlag := fDirectionFlag,
			fThetaStep := fThetaStep,
			bConfigured => bConfigured,
			bBusy => bBusy,
			bPredictionPending => bPredictionPending,
			bPredictionReady => bPredictionReady,
			bResetDone => bResetDone,
			bError => bError,
			nErrorCode => nErrorCode,
			nMaxInferenceDuration => nMaxInferenceDuration,
			aPredictionOutput => aPredictionOutput);
	E_TF3820StandaloneModelId.Model_Wave4_1_Log_Cosh_Robust_Loss:
		fbWave41LogCoshRobustLoss(
			sModelJsonFilePath := 'C:\TwinCAT\3.1\Boot\ML\tf3820\standalone\wave4_1_log_cosh_robust_loss\model.json',
			sMlSvrNetId := sMlSvrNetId,
			eExecutionProvider := eExecutionProvider,
			bEnable := bEnablePrediction,
			bReset := bReset,
			bLoadModel := bLoadSelectedModel,
			nConfigureTimeout := nConfigureTimeout,
			nPredictTimeout := nPredictTimeout,
			nPriority := nPriority,
			fTheta := fTheta,
			fThetaDot := fThetaDot,
			fTorque := fTorque,
			fTemperature := fTemperature,
			fDirectionFlag := fDirectionFlag,
			fThetaStep := fThetaStep,
			bConfigured => bConfigured,
			bBusy => bBusy,
			bPredictionPending => bPredictionPending,
			bPredictionReady => bPredictionReady,
			bResetDone => bResetDone,
			bError => bError,
			nErrorCode => nErrorCode,
			nMaxInferenceDuration => nMaxInferenceDuration,
			aPredictionOutput => aPredictionOutput);
	E_TF3820StandaloneModelId.Model_Wave4_1_Mae_Robust_Loss:
		fbWave41MaeRobustLoss(
			sModelJsonFilePath := 'C:\TwinCAT\3.1\Boot\ML\tf3820\standalone\wave4_1_mae_robust_loss\model.json',
			sMlSvrNetId := sMlSvrNetId,
			eExecutionProvider := eExecutionProvider,
			bEnable := bEnablePrediction,
			bReset := bReset,
			bLoadModel := bLoadSelectedModel,
			nConfigureTimeout := nConfigureTimeout,
			nPredictTimeout := nPredictTimeout,
			nPriority := nPriority,
			fTheta := fTheta,
			fThetaDot := fThetaDot,
			fTorque := fTorque,
			fTemperature := fTemperature,
			fDirectionFlag := fDirectionFlag,
			fThetaStep := fThetaStep,
			bConfigured => bConfigured,
			bBusy => bBusy,
			bPredictionPending => bPredictionPending,
			bPredictionReady => bPredictionReady,
			bResetDone => bResetDone,
			bError => bError,
			nErrorCode => nErrorCode,
			nMaxInferenceDuration => nMaxInferenceDuration,
			aPredictionOutput => aPredictionOutput);
	E_TF3820StandaloneModelId.Model_Wave4_1_Smooth_L1_Robust_Loss:
		fbWave41SmoothL1RobustLoss(
			sModelJsonFilePath := 'C:\TwinCAT\3.1\Boot\ML\tf3820\standalone\wave4_1_smooth_l1_robust_loss\model.json',
			sMlSvrNetId := sMlSvrNetId,
			eExecutionProvider := eExecutionProvider,
			bEnable := bEnablePrediction,
			bReset := bReset,
			bLoadModel := bLoadSelectedModel,
			nConfigureTimeout := nConfigureTimeout,
			nPredictTimeout := nPredictTimeout,
			nPriority := nPriority,
			fTheta := fTheta,
			fThetaDot := fThetaDot,
			fTorque := fTorque,
			fTemperature := fTemperature,
			fDirectionFlag := fDirectionFlag,
			fThetaStep := fThetaStep,
			bConfigured => bConfigured,
			bBusy => bBusy,
			bPredictionPending => bPredictionPending,
			bPredictionReady => bPredictionReady,
			bResetDone => bResetDone,
			bError => bError,
			nErrorCode => nErrorCode,
			nMaxInferenceDuration => nMaxInferenceDuration,
			aPredictionOutput => aPredictionOutput);
	E_TF3820StandaloneModelId.Model_Wave4_2_Gaussian_Nll:
		fbWave42GaussianNll(
			sModelJsonFilePath := 'C:\TwinCAT\3.1\Boot\ML\tf3820\standalone\wave4_2_gaussian_nll\model.json',
			sMlSvrNetId := sMlSvrNetId,
			eExecutionProvider := eExecutionProvider,
			bEnable := bEnablePrediction,
			bReset := bReset,
			bLoadModel := bLoadSelectedModel,
			nConfigureTimeout := nConfigureTimeout,
			nPredictTimeout := nPredictTimeout,
			nPriority := nPriority,
			fTheta := fTheta,
			fThetaDot := fThetaDot,
			fTorque := fTorque,
			fTemperature := fTemperature,
			fDirectionFlag := fDirectionFlag,
			fThetaStep := fThetaStep,
			bConfigured => bConfigured,
			bBusy => bBusy,
			bPredictionPending => bPredictionPending,
			bPredictionReady => bPredictionReady,
			bResetDone => bResetDone,
			bError => bError,
			nErrorCode => nErrorCode,
			nMaxInferenceDuration => nMaxInferenceDuration,
			aPredictionOutput => aPredictionOutput);
	E_TF3820StandaloneModelId.Model_Wave4_2_Quantile_P10_P50_P90:
		fbWave42QuantileP10P50P90(
			sModelJsonFilePath := 'C:\TwinCAT\3.1\Boot\ML\tf3820\standalone\wave4_2_quantile_p10_p50_p90\model.json',
			sMlSvrNetId := sMlSvrNetId,
			eExecutionProvider := eExecutionProvider,
			bEnable := bEnablePrediction,
			bReset := bReset,
			bLoadModel := bLoadSelectedModel,
			nConfigureTimeout := nConfigureTimeout,
			nPredictTimeout := nPredictTimeout,
			nPriority := nPriority,
			fTheta := fTheta,
			fThetaDot := fThetaDot,
			fTorque := fTorque,
			fTemperature := fTemperature,
			fDirectionFlag := fDirectionFlag,
			fThetaStep := fThetaStep,
			bConfigured => bConfigured,
			bBusy => bBusy,
			bPredictionPending => bPredictionPending,
			bPredictionReady => bPredictionReady,
			bResetDone => bResetDone,
			bError => bError,
			nErrorCode => nErrorCode,
			nMaxInferenceDuration => nMaxInferenceDuration,
			aPredictionOutput => aPredictionOutput);
	E_TF3820StandaloneModelId.Model_Wave4_3_Mixture_Density_K2:
		fbWave43MixtureDensityK2(
			sModelJsonFilePath := 'C:\TwinCAT\3.1\Boot\ML\tf3820\standalone\wave4_3_mixture_density_k2\model.json',
			sMlSvrNetId := sMlSvrNetId,
			eExecutionProvider := eExecutionProvider,
			bEnable := bEnablePrediction,
			bReset := bReset,
			bLoadModel := bLoadSelectedModel,
			nConfigureTimeout := nConfigureTimeout,
			nPredictTimeout := nPredictTimeout,
			nPriority := nPriority,
			fTheta := fTheta,
			fThetaDot := fThetaDot,
			fTorque := fTorque,
			fTemperature := fTemperature,
			fDirectionFlag := fDirectionFlag,
			fThetaStep := fThetaStep,
			bConfigured => bConfigured,
			bBusy => bBusy,
			bPredictionPending => bPredictionPending,
			bPredictionReady => bPredictionReady,
			bResetDone => bResetDone,
			bError => bError,
			nErrorCode => nErrorCode,
			nMaxInferenceDuration => nMaxInferenceDuration,
			aPredictionOutput => aPredictionOutput);
	E_TF3820StandaloneModelId.Model_Wave4_3_Mixture_Density_K3:
		fbWave43MixtureDensityK3(
			sModelJsonFilePath := 'C:\TwinCAT\3.1\Boot\ML\tf3820\standalone\wave4_3_mixture_density_k3\model.json',
			sMlSvrNetId := sMlSvrNetId,
			eExecutionProvider := eExecutionProvider,
			bEnable := bEnablePrediction,
			bReset := bReset,
			bLoadModel := bLoadSelectedModel,
			nConfigureTimeout := nConfigureTimeout,
			nPredictTimeout := nPredictTimeout,
			nPriority := nPriority,
			fTheta := fTheta,
			fThetaDot := fThetaDot,
			fTorque := fTorque,
			fTemperature := fTemperature,
			fDirectionFlag := fDirectionFlag,
			fThetaStep := fThetaStep,
			bConfigured => bConfigured,
			bBusy => bBusy,
			bPredictionPending => bPredictionPending,
			bPredictionReady => bPredictionReady,
			bResetDone => bResetDone,
			bError => bError,
			nErrorCode => nErrorCode,
			nMaxInferenceDuration => nMaxInferenceDuration,
			aPredictionOutput => aPredictionOutput);
	E_TF3820StandaloneModelId.Model_Wave4_4_Causal_Tcn_Latent_Offset_Residual:
		fbWave44CausalTcnLatentOffsetResidual(
			sModelJsonFilePath := 'C:\TwinCAT\3.1\Boot\ML\tf3820\standalone\wave4_4_causal_tcn_latent_offset_residual\model.json',
			sMlSvrNetId := sMlSvrNetId,
			eExecutionProvider := eExecutionProvider,
			bEnable := bEnablePrediction,
			bReset := bReset,
			bLoadModel := bLoadSelectedModel,
			nConfigureTimeout := nConfigureTimeout,
			nPredictTimeout := nPredictTimeout,
			nPriority := nPriority,
			fTheta := fTheta,
			fThetaDot := fThetaDot,
			fTorque := fTorque,
			fTemperature := fTemperature,
			fDirectionFlag := fDirectionFlag,
			fThetaStep := fThetaStep,
			bConfigured => bConfigured,
			bBusy => bBusy,
			bPredictionPending => bPredictionPending,
			bPredictionReady => bPredictionReady,
			bResetDone => bResetDone,
			bError => bError,
			nErrorCode => nErrorCode,
			nMaxInferenceDuration => nMaxInferenceDuration,
			aPredictionOutput => aPredictionOutput);
	E_TF3820StandaloneModelId.Model_Wave4_4_Gru_Latent_Offset_Residual:
		fbWave44GruLatentOffsetResidual(
			sModelJsonFilePath := 'C:\TwinCAT\3.1\Boot\ML\tf3820\standalone\wave4_4_gru_latent_offset_residual\model.json',
			sMlSvrNetId := sMlSvrNetId,
			eExecutionProvider := eExecutionProvider,
			bEnable := bEnablePrediction,
			bReset := bReset,
			bLoadModel := bLoadSelectedModel,
			nConfigureTimeout := nConfigureTimeout,
			nPredictTimeout := nPredictTimeout,
			nPriority := nPriority,
			fTheta := fTheta,
			fThetaDot := fThetaDot,
			fTorque := fTorque,
			fTemperature := fTemperature,
			fDirectionFlag := fDirectionFlag,
			fThetaStep := fThetaStep,
			bConfigured => bConfigured,
			bBusy => bBusy,
			bPredictionPending => bPredictionPending,
			bPredictionReady => bPredictionReady,
			bResetDone => bResetDone,
			bError => bError,
			nErrorCode => nErrorCode,
			nMaxInferenceDuration => nMaxInferenceDuration,
			aPredictionOutput => aPredictionOutput);
	E_TF3820StandaloneModelId.Model_Wave5_1_Harmonic_Prior_Pointwise_Control:
		fbWave51HarmonicPriorPointwiseControl(
			sModelJsonFilePath := 'C:\TwinCAT\3.1\Boot\ML\tf3820\standalone\wave5_1_harmonic_prior_pointwise_control\model.json',
			sMlSvrNetId := sMlSvrNetId,
			eExecutionProvider := eExecutionProvider,
			bEnable := bEnablePrediction,
			bReset := bReset,
			bLoadModel := bLoadSelectedModel,
			nConfigureTimeout := nConfigureTimeout,
			nPredictTimeout := nPredictTimeout,
			nPriority := nPriority,
			fTheta := fTheta,
			fThetaDot := fThetaDot,
			fTorque := fTorque,
			fTemperature := fTemperature,
			fDirectionFlag := fDirectionFlag,
			fThetaStep := fThetaStep,
			bConfigured => bConfigured,
			bBusy => bBusy,
			bPredictionPending => bPredictionPending,
			bPredictionReady => bPredictionReady,
			bResetDone => bResetDone,
			bError => bError,
			nErrorCode => nErrorCode,
			nMaxInferenceDuration => nMaxInferenceDuration,
			aPredictionOutput => aPredictionOutput);
	E_TF3820StandaloneModelId.Model_Wave5_1_Harmonic_Prior_Smooth_L1_Structured:
		fbWave51HarmonicPriorSmoothL1Structured(
			sModelJsonFilePath := 'C:\TwinCAT\3.1\Boot\ML\tf3820\standalone\wave5_1_harmonic_prior_smooth_l1_structured\model.json',
			sMlSvrNetId := sMlSvrNetId,
			eExecutionProvider := eExecutionProvider,
			bEnable := bEnablePrediction,
			bReset := bReset,
			bLoadModel := bLoadSelectedModel,
			nConfigureTimeout := nConfigureTimeout,
			nPredictTimeout := nPredictTimeout,
			nPriority := nPriority,
			fTheta := fTheta,
			fThetaDot := fThetaDot,
			fTorque := fTorque,
			fTemperature := fTemperature,
			fDirectionFlag := fDirectionFlag,
			fThetaStep := fThetaStep,
			bConfigured => bConfigured,
			bBusy => bBusy,
			bPredictionPending => bPredictionPending,
			bPredictionReady => bPredictionReady,
			bResetDone => bResetDone,
			bError => bError,
			nErrorCode => nErrorCode,
			nMaxInferenceDuration => nMaxInferenceDuration,
			aPredictionOutput => aPredictionOutput);
END_CASE

END_PROGRAM

// ---- POUs/FB_FeedforwardTf3820Runner.TcPOU
FUNCTION_BLOCK FB_FeedforwardTf3820Runner
VAR_INPUT
	sModelJsonFilePath	: T_MaxString;
	sMlSvrNetId			: T_MaxString := 'local';
	eExecutionProvider	: E_ExecutionProvider := E_ExecutionProvider.CPU;
	bEnable				: BOOL;
	bReset					: BOOL;
	bLoadModel			: BOOL;
	nConfigureTimeout	: UDINT := 1000;
	nPredictTimeout		: UDINT := 100;
	nPriority			: UDINT := 0;
	fTheta					: REAL;
	fThetaDot				: REAL;
	fTorque				: REAL;
	fTemperature			: REAL;
	fDirectionFlag		: REAL;
	fThetaStep			: REAL := 0.25;
END_VAR
VAR
	fbMlSvr				: FB_MlSvrPrediction;
	stModelInput		: ST_FeedforwardInput;
	stModelOutput		: ST_FeedforwardOutput;
	rtrig_model			: R_TRIG;
	nState					: INT := 0;
	nSequenceIndex		: INT;
	nOutputIndex		: INT;
END_VAR
VAR_OUTPUT
	bConfigured			: BOOL;
	bBusy					: BOOL;
	bPredictionPending	: BOOL;
	bPredictionReady	: BOOL;
	bResetDone			: BOOL;
	bError					: BOOL;
	nErrorCode			: HRESULT;
	nMaxInferenceDuration	: UDINT;
	aPredictionOutput	: ARRAY[0..8] OF REAL;
END_VAR

rtrig_model(CLK := bLoadModel);

IF rtrig_model.Q THEN
	bPredictionPending := FALSE;
	bPredictionReady := FALSE;
	bResetDone := FALSE;
	bError := FALSE;
	IF fbMlSvr.bConfigured THEN
		nState := 5;
	ELSE
		bConfigured := FALSE;
		nState := 10;
	END_IF
END_IF

IF bReset THEN
	bPredictionPending := FALSE;
	bPredictionReady := FALSE;
	bError := FALSE;
	IF fbMlSvr.bConfigured THEN
		nState := 5;
	ELSE
		bConfigured := FALSE;
		bResetDone := TRUE;
		nState := 0;
	END_IF
END_IF

CASE nState OF
	0:
		bBusy := FALSE;
		IF bLoadModel AND NOT(bConfigured) AND NOT(bReset) THEN
			nState := 10;
		END_IF

	5:
		bBusy := TRUE;
		IF fbMlSvr.Deconfigure(nTimeout := nConfigureTimeout) THEN
			nErrorCode := fbMlSvr.nErrorCode;
			bError := fbMlSvr.bError OR (nErrorCode <> 0);
			bConfigured := FALSE;
			bBusy := FALSE;
			bResetDone := NOT(bError);
			IF bError THEN
				nState := 90;
			ELSIF bReset THEN
				nState := 0;
			ELSE
				nState := 10;
			END_IF
		END_IF

	10:
		bBusy := TRUE;
		fbMlSvr.stPredictionParameter.sMlModelFilePath := sModelJsonFilePath;
		fbMlSvr.stPredictionParameter.sMlSvrNetId := sMlSvrNetId;
		fbMlSvr.stPredictionParameter.eExecutionProvider := eExecutionProvider;
		IF fbMlSvr.Configure(nTimeout := nConfigureTimeout, nPriority := nPriority) THEN
			nErrorCode := fbMlSvr.nErrorCode;
			bError := fbMlSvr.bError OR (nErrorCode <> 0);
			bConfigured := fbMlSvr.bConfigured AND NOT(bError);
			bBusy := FALSE;
			IF bConfigured THEN
				nState := 20;
			ELSE
				nState := 90;
			END_IF
		END_IF

	20:
		bBusy := FALSE;
		bPredictionPending := FALSE;
		IF bEnable AND bConfigured AND NOT(bError) AND NOT(bReset) THEN
			stModelInput.in_input_tensor[0,0] := fTheta;
			stModelInput.in_input_tensor[0,1] := fThetaDot;
			stModelInput.in_input_tensor[0,2] := fTorque;
			stModelInput.in_input_tensor[0,3] := fTemperature;
			stModelInput.in_input_tensor[0,4] := fDirectionFlag;
			bPredictionReady := FALSE;
			bPredictionPending := TRUE;
			nState := 30;
		END_IF

	30:
		bBusy := TRUE;
		bPredictionPending := TRUE;
		IF fbMlSvr.Predict(
			pDataIn := ADR(stModelInput),
			nDataInSize := SIZEOF(ST_FeedforwardInput),
			pDataOut := ADR(stModelOutput),
			nDataOutSize := SIZEOF(ST_FeedforwardOutput),
			nTimeout := nPredictTimeout,
			nPriority := nPriority) THEN
			nErrorCode := fbMlSvr.nErrorCode;
			bError := fbMlSvr.bError OR (nErrorCode <> 0);
			nMaxInferenceDuration := fbMlSvr.nMaxInferenceDuration;
			bPredictionPending := FALSE;
			bBusy := FALSE;
			IF NOT(bError) THEN
				aPredictionOutput[0] := stModelOutput.out_prediction_tensor[0,0];
				FOR nOutputIndex := 1 TO 8 DO
					aPredictionOutput[nOutputIndex] := 0.0;
				END_FOR
				bPredictionReady := TRUE;
				nState := 20;
			ELSE
				nState := 90;
			END_IF
		END_IF

	90:
		bBusy := FALSE;
		bPredictionPending := FALSE;
		bError := TRUE;
END_CASE

nErrorCode := fbMlSvr.nErrorCode;
nMaxInferenceDuration := fbMlSvr.nMaxInferenceDuration;

END_FUNCTION_BLOCK

// ---- POUs/FB_GruSequenceTf3820Runner.TcPOU
FUNCTION_BLOCK FB_GruSequenceTf3820Runner
VAR_INPUT
	sModelJsonFilePath	: T_MaxString;
	sMlSvrNetId			: T_MaxString := 'local';
	eExecutionProvider	: E_ExecutionProvider := E_ExecutionProvider.CPU;
	bEnable				: BOOL;
	bReset					: BOOL;
	bLoadModel			: BOOL;
	nConfigureTimeout	: UDINT := 1000;
	nPredictTimeout		: UDINT := 100;
	nPriority			: UDINT := 0;
	fTheta					: REAL;
	fThetaDot				: REAL;
	fTorque				: REAL;
	fTemperature			: REAL;
	fDirectionFlag		: REAL;
	fThetaStep			: REAL := 0.25;
END_VAR
VAR
	fbMlSvr				: FB_MlSvrPrediction;
	stModelInput		: ST_GruSequenceInput;
	stModelOutput		: ST_GruSequenceOutput;
	rtrig_model			: R_TRIG;
	nState					: INT := 0;
	nSequenceIndex		: INT;
	nOutputIndex		: INT;
END_VAR
VAR_OUTPUT
	bConfigured			: BOOL;
	bBusy					: BOOL;
	bPredictionPending	: BOOL;
	bPredictionReady	: BOOL;
	bResetDone			: BOOL;
	bError					: BOOL;
	nErrorCode			: HRESULT;
	nMaxInferenceDuration	: UDINT;
	aPredictionOutput	: ARRAY[0..8] OF REAL;
END_VAR

rtrig_model(CLK := bLoadModel);

IF rtrig_model.Q THEN
	bPredictionPending := FALSE;
	bPredictionReady := FALSE;
	bResetDone := FALSE;
	bError := FALSE;
	IF fbMlSvr.bConfigured THEN
		nState := 5;
	ELSE
		bConfigured := FALSE;
		nState := 10;
	END_IF
END_IF

IF bReset THEN
	bPredictionPending := FALSE;
	bPredictionReady := FALSE;
	bError := FALSE;
	IF fbMlSvr.bConfigured THEN
		nState := 5;
	ELSE
		bConfigured := FALSE;
		bResetDone := TRUE;
		nState := 0;
	END_IF
END_IF

CASE nState OF
	0:
		bBusy := FALSE;
		IF bLoadModel AND NOT(bConfigured) AND NOT(bReset) THEN
			nState := 10;
		END_IF

	5:
		bBusy := TRUE;
		IF fbMlSvr.Deconfigure(nTimeout := nConfigureTimeout) THEN
			nErrorCode := fbMlSvr.nErrorCode;
			bError := fbMlSvr.bError OR (nErrorCode <> 0);
			bConfigured := FALSE;
			bBusy := FALSE;
			bResetDone := NOT(bError);
			IF bError THEN
				nState := 90;
			ELSIF bReset THEN
				nState := 0;
			ELSE
				nState := 10;
			END_IF
		END_IF

	10:
		bBusy := TRUE;
		fbMlSvr.stPredictionParameter.sMlModelFilePath := sModelJsonFilePath;
		fbMlSvr.stPredictionParameter.sMlSvrNetId := sMlSvrNetId;
		fbMlSvr.stPredictionParameter.eExecutionProvider := eExecutionProvider;
		IF fbMlSvr.Configure(nTimeout := nConfigureTimeout, nPriority := nPriority) THEN
			nErrorCode := fbMlSvr.nErrorCode;
			bError := fbMlSvr.bError OR (nErrorCode <> 0);
			bConfigured := fbMlSvr.bConfigured AND NOT(bError);
			bBusy := FALSE;
			IF bConfigured THEN
				nState := 20;
			ELSE
				nState := 90;
			END_IF
		END_IF

	20:
		bBusy := FALSE;
		bPredictionPending := FALSE;
		IF bEnable AND bConfigured AND NOT(bError) AND NOT(bReset) THEN
			FOR nSequenceIndex := 0 TO 32 DO
				stModelInput.in_input_tensor[0,nSequenceIndex,0] := fTheta + (INT_TO_REAL(nSequenceIndex) * fThetaStep);
				stModelInput.in_input_tensor[0,nSequenceIndex,1] := fThetaDot;
				stModelInput.in_input_tensor[0,nSequenceIndex,2] := fTorque;
				stModelInput.in_input_tensor[0,nSequenceIndex,3] := fTemperature;
				stModelInput.in_input_tensor[0,nSequenceIndex,4] := fDirectionFlag;
			END_FOR
			bPredictionReady := FALSE;
			bPredictionPending := TRUE;
			nState := 30;
		END_IF

	30:
		bBusy := TRUE;
		bPredictionPending := TRUE;
		IF fbMlSvr.Predict(
			pDataIn := ADR(stModelInput),
			nDataInSize := SIZEOF(ST_GruSequenceInput),
			pDataOut := ADR(stModelOutput),
			nDataOutSize := SIZEOF(ST_GruSequenceOutput),
			nTimeout := nPredictTimeout,
			nPriority := nPriority) THEN
			nErrorCode := fbMlSvr.nErrorCode;
			bError := fbMlSvr.bError OR (nErrorCode <> 0);
			nMaxInferenceDuration := fbMlSvr.nMaxInferenceDuration;
			bPredictionPending := FALSE;
			bBusy := FALSE;
			IF NOT(bError) THEN
				aPredictionOutput[0] := stModelOutput.out_prediction_tensor[0,0];
				FOR nOutputIndex := 1 TO 8 DO
					aPredictionOutput[nOutputIndex] := 0.0;
				END_FOR
				bPredictionReady := TRUE;
				nState := 20;
			ELSE
				nState := 90;
			END_IF
		END_IF

	90:
		bBusy := FALSE;
		bPredictionPending := FALSE;
		bError := TRUE;
END_CASE

nErrorCode := fbMlSvr.nErrorCode;
nMaxInferenceDuration := fbMlSvr.nMaxInferenceDuration;

END_FUNCTION_BLOCK

// ---- POUs/FB_HarmonicRegressionTf3820Runner.TcPOU
FUNCTION_BLOCK FB_HarmonicRegressionTf3820Runner
VAR_INPUT
	sModelJsonFilePath	: T_MaxString;
	sMlSvrNetId			: T_MaxString := 'local';
	eExecutionProvider	: E_ExecutionProvider := E_ExecutionProvider.CPU;
	bEnable				: BOOL;
	bReset					: BOOL;
	bLoadModel			: BOOL;
	nConfigureTimeout	: UDINT := 1000;
	nPredictTimeout		: UDINT := 100;
	nPriority			: UDINT := 0;
	fTheta					: REAL;
	fThetaDot				: REAL;
	fTorque				: REAL;
	fTemperature			: REAL;
	fDirectionFlag		: REAL;
	fThetaStep			: REAL := 0.25;
END_VAR
VAR
	fbMlSvr				: FB_MlSvrPrediction;
	stModelInput		: ST_HarmonicRegressionInput;
	stModelOutput		: ST_HarmonicRegressionOutput;
	rtrig_model			: R_TRIG;
	nState					: INT := 0;
	nSequenceIndex		: INT;
	nOutputIndex		: INT;
END_VAR
VAR_OUTPUT
	bConfigured			: BOOL;
	bBusy					: BOOL;
	bPredictionPending	: BOOL;
	bPredictionReady	: BOOL;
	bResetDone			: BOOL;
	bError					: BOOL;
	nErrorCode			: HRESULT;
	nMaxInferenceDuration	: UDINT;
	aPredictionOutput	: ARRAY[0..8] OF REAL;
END_VAR

rtrig_model(CLK := bLoadModel);

IF rtrig_model.Q THEN
	bPredictionPending := FALSE;
	bPredictionReady := FALSE;
	bResetDone := FALSE;
	bError := FALSE;
	IF fbMlSvr.bConfigured THEN
		nState := 5;
	ELSE
		bConfigured := FALSE;
		nState := 10;
	END_IF
END_IF

IF bReset THEN
	bPredictionPending := FALSE;
	bPredictionReady := FALSE;
	bError := FALSE;
	IF fbMlSvr.bConfigured THEN
		nState := 5;
	ELSE
		bConfigured := FALSE;
		bResetDone := TRUE;
		nState := 0;
	END_IF
END_IF

CASE nState OF
	0:
		bBusy := FALSE;
		IF bLoadModel AND NOT(bConfigured) AND NOT(bReset) THEN
			nState := 10;
		END_IF

	5:
		bBusy := TRUE;
		IF fbMlSvr.Deconfigure(nTimeout := nConfigureTimeout) THEN
			nErrorCode := fbMlSvr.nErrorCode;
			bError := fbMlSvr.bError OR (nErrorCode <> 0);
			bConfigured := FALSE;
			bBusy := FALSE;
			bResetDone := NOT(bError);
			IF bError THEN
				nState := 90;
			ELSIF bReset THEN
				nState := 0;
			ELSE
				nState := 10;
			END_IF
		END_IF

	10:
		bBusy := TRUE;
		fbMlSvr.stPredictionParameter.sMlModelFilePath := sModelJsonFilePath;
		fbMlSvr.stPredictionParameter.sMlSvrNetId := sMlSvrNetId;
		fbMlSvr.stPredictionParameter.eExecutionProvider := eExecutionProvider;
		IF fbMlSvr.Configure(nTimeout := nConfigureTimeout, nPriority := nPriority) THEN
			nErrorCode := fbMlSvr.nErrorCode;
			bError := fbMlSvr.bError OR (nErrorCode <> 0);
			bConfigured := fbMlSvr.bConfigured AND NOT(bError);
			bBusy := FALSE;
			IF bConfigured THEN
				nState := 20;
			ELSE
				nState := 90;
			END_IF
		END_IF

	20:
		bBusy := FALSE;
		bPredictionPending := FALSE;
		IF bEnable AND bConfigured AND NOT(bError) AND NOT(bReset) THEN
			stModelInput.in_input_tensor[0,0] := fTheta;
			stModelInput.in_input_tensor[0,1] := fThetaDot;
			stModelInput.in_input_tensor[0,2] := fTorque;
			stModelInput.in_input_tensor[0,3] := fTemperature;
			stModelInput.in_input_tensor[0,4] := fDirectionFlag;
			bPredictionReady := FALSE;
			bPredictionPending := TRUE;
			nState := 30;
		END_IF

	30:
		bBusy := TRUE;
		bPredictionPending := TRUE;
		IF fbMlSvr.Predict(
			pDataIn := ADR(stModelInput),
			nDataInSize := SIZEOF(ST_HarmonicRegressionInput),
			pDataOut := ADR(stModelOutput),
			nDataOutSize := SIZEOF(ST_HarmonicRegressionOutput),
			nTimeout := nPredictTimeout,
			nPriority := nPriority) THEN
			nErrorCode := fbMlSvr.nErrorCode;
			bError := fbMlSvr.bError OR (nErrorCode <> 0);
			nMaxInferenceDuration := fbMlSvr.nMaxInferenceDuration;
			bPredictionPending := FALSE;
			bBusy := FALSE;
			IF NOT(bError) THEN
				aPredictionOutput[0] := stModelOutput.out_prediction_tensor[0,0];
				FOR nOutputIndex := 1 TO 8 DO
					aPredictionOutput[nOutputIndex] := 0.0;
				END_FOR
				bPredictionReady := TRUE;
				nState := 20;
			ELSE
				nState := 90;
			END_IF
		END_IF

	90:
		bBusy := FALSE;
		bPredictionPending := FALSE;
		bError := TRUE;
END_CASE

nErrorCode := fbMlSvr.nErrorCode;
nMaxInferenceDuration := fbMlSvr.nMaxInferenceDuration;

END_FUNCTION_BLOCK

// ---- POUs/FB_LstmSequenceTf3820Runner.TcPOU
FUNCTION_BLOCK FB_LstmSequenceTf3820Runner
VAR_INPUT
	sModelJsonFilePath	: T_MaxString;
	sMlSvrNetId			: T_MaxString := 'local';
	eExecutionProvider	: E_ExecutionProvider := E_ExecutionProvider.CPU;
	bEnable				: BOOL;
	bReset					: BOOL;
	bLoadModel			: BOOL;
	nConfigureTimeout	: UDINT := 1000;
	nPredictTimeout		: UDINT := 100;
	nPriority			: UDINT := 0;
	fTheta					: REAL;
	fThetaDot				: REAL;
	fTorque				: REAL;
	fTemperature			: REAL;
	fDirectionFlag		: REAL;
	fThetaStep			: REAL := 0.25;
END_VAR
VAR
	fbMlSvr				: FB_MlSvrPrediction;
	stModelInput		: ST_LstmSequenceInput;
	stModelOutput		: ST_LstmSequenceOutput;
	rtrig_model			: R_TRIG;
	nState					: INT := 0;
	nSequenceIndex		: INT;
	nOutputIndex		: INT;
END_VAR
VAR_OUTPUT
	bConfigured			: BOOL;
	bBusy					: BOOL;
	bPredictionPending	: BOOL;
	bPredictionReady	: BOOL;
	bResetDone			: BOOL;
	bError					: BOOL;
	nErrorCode			: HRESULT;
	nMaxInferenceDuration	: UDINT;
	aPredictionOutput	: ARRAY[0..8] OF REAL;
END_VAR

rtrig_model(CLK := bLoadModel);

IF rtrig_model.Q THEN
	bPredictionPending := FALSE;
	bPredictionReady := FALSE;
	bResetDone := FALSE;
	bError := FALSE;
	IF fbMlSvr.bConfigured THEN
		nState := 5;
	ELSE
		bConfigured := FALSE;
		nState := 10;
	END_IF
END_IF

IF bReset THEN
	bPredictionPending := FALSE;
	bPredictionReady := FALSE;
	bError := FALSE;
	IF fbMlSvr.bConfigured THEN
		nState := 5;
	ELSE
		bConfigured := FALSE;
		bResetDone := TRUE;
		nState := 0;
	END_IF
END_IF

CASE nState OF
	0:
		bBusy := FALSE;
		IF bLoadModel AND NOT(bConfigured) AND NOT(bReset) THEN
			nState := 10;
		END_IF

	5:
		bBusy := TRUE;
		IF fbMlSvr.Deconfigure(nTimeout := nConfigureTimeout) THEN
			nErrorCode := fbMlSvr.nErrorCode;
			bError := fbMlSvr.bError OR (nErrorCode <> 0);
			bConfigured := FALSE;
			bBusy := FALSE;
			bResetDone := NOT(bError);
			IF bError THEN
				nState := 90;
			ELSIF bReset THEN
				nState := 0;
			ELSE
				nState := 10;
			END_IF
		END_IF

	10:
		bBusy := TRUE;
		fbMlSvr.stPredictionParameter.sMlModelFilePath := sModelJsonFilePath;
		fbMlSvr.stPredictionParameter.sMlSvrNetId := sMlSvrNetId;
		fbMlSvr.stPredictionParameter.eExecutionProvider := eExecutionProvider;
		IF fbMlSvr.Configure(nTimeout := nConfigureTimeout, nPriority := nPriority) THEN
			nErrorCode := fbMlSvr.nErrorCode;
			bError := fbMlSvr.bError OR (nErrorCode <> 0);
			bConfigured := fbMlSvr.bConfigured AND NOT(bError);
			bBusy := FALSE;
			IF bConfigured THEN
				nState := 20;
			ELSE
				nState := 90;
			END_IF
		END_IF

	20:
		bBusy := FALSE;
		bPredictionPending := FALSE;
		IF bEnable AND bConfigured AND NOT(bError) AND NOT(bReset) THEN
			FOR nSequenceIndex := 0 TO 32 DO
				stModelInput.in_input_tensor[0,nSequenceIndex,0] := fTheta + (INT_TO_REAL(nSequenceIndex) * fThetaStep);
				stModelInput.in_input_tensor[0,nSequenceIndex,1] := fThetaDot;
				stModelInput.in_input_tensor[0,nSequenceIndex,2] := fTorque;
				stModelInput.in_input_tensor[0,nSequenceIndex,3] := fTemperature;
				stModelInput.in_input_tensor[0,nSequenceIndex,4] := fDirectionFlag;
			END_FOR
			bPredictionReady := FALSE;
			bPredictionPending := TRUE;
			nState := 30;
		END_IF

	30:
		bBusy := TRUE;
		bPredictionPending := TRUE;
		IF fbMlSvr.Predict(
			pDataIn := ADR(stModelInput),
			nDataInSize := SIZEOF(ST_LstmSequenceInput),
			pDataOut := ADR(stModelOutput),
			nDataOutSize := SIZEOF(ST_LstmSequenceOutput),
			nTimeout := nPredictTimeout,
			nPriority := nPriority) THEN
			nErrorCode := fbMlSvr.nErrorCode;
			bError := fbMlSvr.bError OR (nErrorCode <> 0);
			nMaxInferenceDuration := fbMlSvr.nMaxInferenceDuration;
			bPredictionPending := FALSE;
			bBusy := FALSE;
			IF NOT(bError) THEN
				aPredictionOutput[0] := stModelOutput.out_prediction_tensor[0,0];
				FOR nOutputIndex := 1 TO 8 DO
					aPredictionOutput[nOutputIndex] := 0.0;
				END_FOR
				bPredictionReady := TRUE;
				nState := 20;
			ELSE
				nState := 90;
			END_IF
		END_IF

	90:
		bBusy := FALSE;
		bPredictionPending := FALSE;
		bError := TRUE;
END_CASE

nErrorCode := fbMlSvr.nErrorCode;
nMaxInferenceDuration := fbMlSvr.nMaxInferenceDuration;

END_FUNCTION_BLOCK

// ---- POUs/FB_PeriodicGruSequenceTf3820Runner.TcPOU
FUNCTION_BLOCK FB_PeriodicGruSequenceTf3820Runner
VAR_INPUT
	sModelJsonFilePath	: T_MaxString;
	sMlSvrNetId			: T_MaxString := 'local';
	eExecutionProvider	: E_ExecutionProvider := E_ExecutionProvider.CPU;
	bEnable				: BOOL;
	bReset					: BOOL;
	bLoadModel			: BOOL;
	nConfigureTimeout	: UDINT := 1000;
	nPredictTimeout		: UDINT := 100;
	nPriority			: UDINT := 0;
	fTheta					: REAL;
	fThetaDot				: REAL;
	fTorque				: REAL;
	fTemperature			: REAL;
	fDirectionFlag		: REAL;
	fThetaStep			: REAL := 0.25;
END_VAR
VAR
	fbMlSvr				: FB_MlSvrPrediction;
	stModelInput		: ST_PeriodicGruSequenceInput;
	stModelOutput		: ST_PeriodicGruSequenceOutput;
	rtrig_model			: R_TRIG;
	nState					: INT := 0;
	nSequenceIndex		: INT;
	nOutputIndex		: INT;
END_VAR
VAR_OUTPUT
	bConfigured			: BOOL;
	bBusy					: BOOL;
	bPredictionPending	: BOOL;
	bPredictionReady	: BOOL;
	bResetDone			: BOOL;
	bError					: BOOL;
	nErrorCode			: HRESULT;
	nMaxInferenceDuration	: UDINT;
	aPredictionOutput	: ARRAY[0..8] OF REAL;
END_VAR

rtrig_model(CLK := bLoadModel);

IF rtrig_model.Q THEN
	bPredictionPending := FALSE;
	bPredictionReady := FALSE;
	bResetDone := FALSE;
	bError := FALSE;
	IF fbMlSvr.bConfigured THEN
		nState := 5;
	ELSE
		bConfigured := FALSE;
		nState := 10;
	END_IF
END_IF

IF bReset THEN
	bPredictionPending := FALSE;
	bPredictionReady := FALSE;
	bError := FALSE;
	IF fbMlSvr.bConfigured THEN
		nState := 5;
	ELSE
		bConfigured := FALSE;
		bResetDone := TRUE;
		nState := 0;
	END_IF
END_IF

CASE nState OF
	0:
		bBusy := FALSE;
		IF bLoadModel AND NOT(bConfigured) AND NOT(bReset) THEN
			nState := 10;
		END_IF

	5:
		bBusy := TRUE;
		IF fbMlSvr.Deconfigure(nTimeout := nConfigureTimeout) THEN
			nErrorCode := fbMlSvr.nErrorCode;
			bError := fbMlSvr.bError OR (nErrorCode <> 0);
			bConfigured := FALSE;
			bBusy := FALSE;
			bResetDone := NOT(bError);
			IF bError THEN
				nState := 90;
			ELSIF bReset THEN
				nState := 0;
			ELSE
				nState := 10;
			END_IF
		END_IF

	10:
		bBusy := TRUE;
		fbMlSvr.stPredictionParameter.sMlModelFilePath := sModelJsonFilePath;
		fbMlSvr.stPredictionParameter.sMlSvrNetId := sMlSvrNetId;
		fbMlSvr.stPredictionParameter.eExecutionProvider := eExecutionProvider;
		IF fbMlSvr.Configure(nTimeout := nConfigureTimeout, nPriority := nPriority) THEN
			nErrorCode := fbMlSvr.nErrorCode;
			bError := fbMlSvr.bError OR (nErrorCode <> 0);
			bConfigured := fbMlSvr.bConfigured AND NOT(bError);
			bBusy := FALSE;
			IF bConfigured THEN
				nState := 20;
			ELSE
				nState := 90;
			END_IF
		END_IF

	20:
		bBusy := FALSE;
		bPredictionPending := FALSE;
		IF bEnable AND bConfigured AND NOT(bError) AND NOT(bReset) THEN
			FOR nSequenceIndex := 0 TO 32 DO
				stModelInput.in_input_tensor[0,nSequenceIndex,0] := fTheta + (INT_TO_REAL(nSequenceIndex) * fThetaStep);
				stModelInput.in_input_tensor[0,nSequenceIndex,1] := fThetaDot;
				stModelInput.in_input_tensor[0,nSequenceIndex,2] := fTorque;
				stModelInput.in_input_tensor[0,nSequenceIndex,3] := fTemperature;
				stModelInput.in_input_tensor[0,nSequenceIndex,4] := fDirectionFlag;
			END_FOR
			bPredictionReady := FALSE;
			bPredictionPending := TRUE;
			nState := 30;
		END_IF

	30:
		bBusy := TRUE;
		bPredictionPending := TRUE;
		IF fbMlSvr.Predict(
			pDataIn := ADR(stModelInput),
			nDataInSize := SIZEOF(ST_PeriodicGruSequenceInput),
			pDataOut := ADR(stModelOutput),
			nDataOutSize := SIZEOF(ST_PeriodicGruSequenceOutput),
			nTimeout := nPredictTimeout,
			nPriority := nPriority) THEN
			nErrorCode := fbMlSvr.nErrorCode;
			bError := fbMlSvr.bError OR (nErrorCode <> 0);
			nMaxInferenceDuration := fbMlSvr.nMaxInferenceDuration;
			bPredictionPending := FALSE;
			bBusy := FALSE;
			IF NOT(bError) THEN
				aPredictionOutput[0] := stModelOutput.out_prediction_tensor[0,0];
				FOR nOutputIndex := 1 TO 8 DO
					aPredictionOutput[nOutputIndex] := 0.0;
				END_FOR
				bPredictionReady := TRUE;
				nState := 20;
			ELSE
				nState := 90;
			END_IF
		END_IF

	90:
		bBusy := FALSE;
		bPredictionPending := FALSE;
		bError := TRUE;
END_CASE

